// Mitsubishi GX Works2 project: GOL-923VNW-21110019(220112)   PLC: Q02U

PROGRAM OVEN
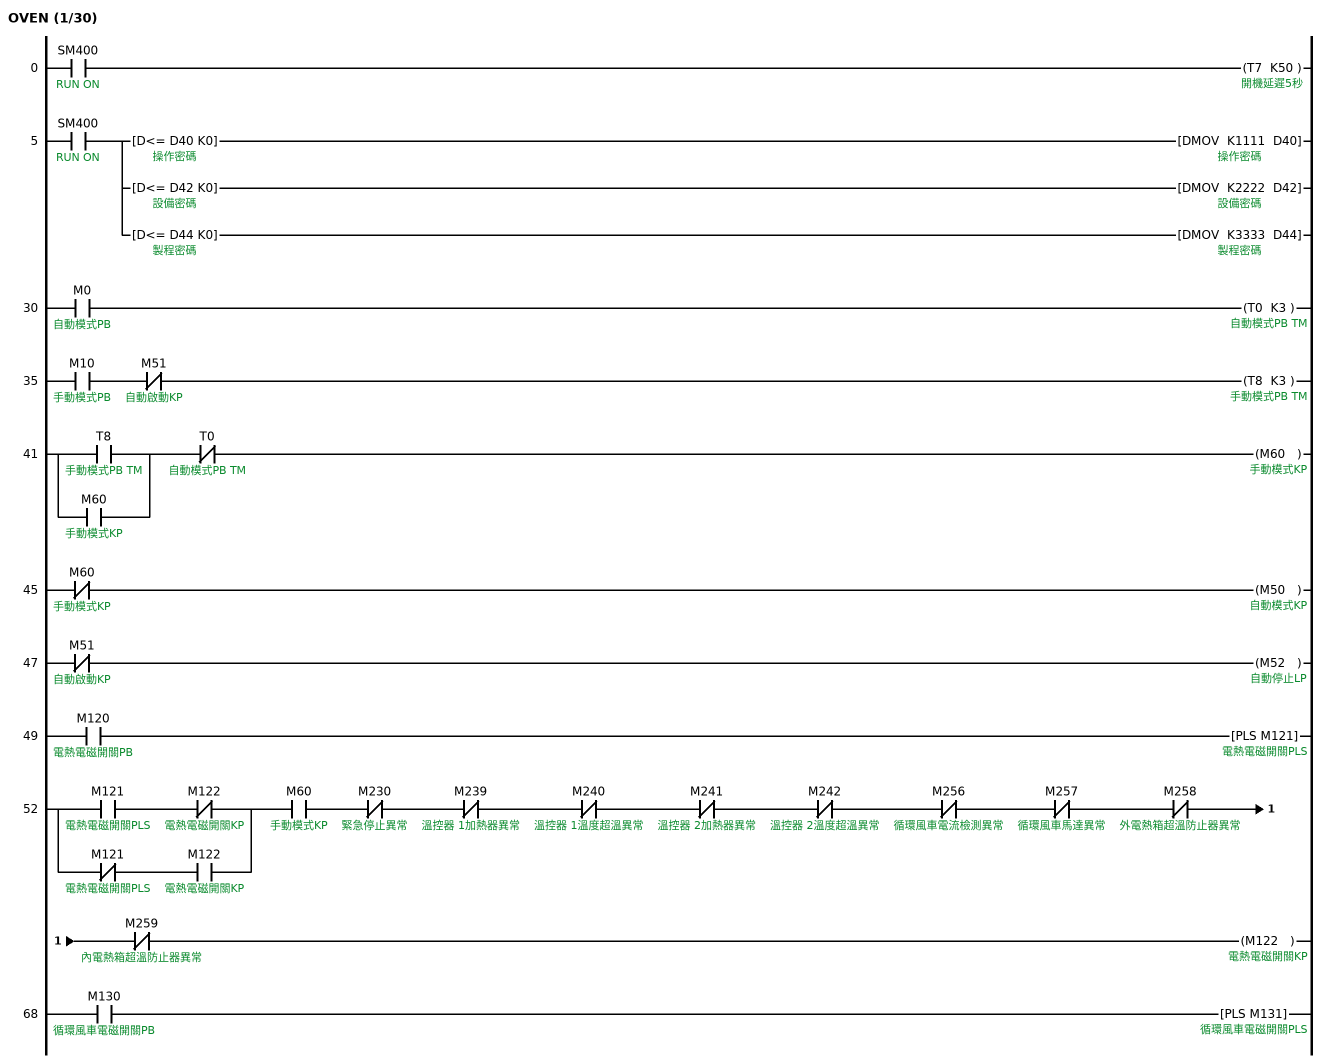
0     LD      SM400  ; RUN ON
      OUT     T7 K50  ; 開機延遲5秒
5     LD      SM400  ; RUN ON
      MPS
      ANDD<=  D40 K0  ; 操作密碼
      DMOV    K1111 D40
      MRD
      ANDD<=  D42 K0  ; 設備密碼
      DMOV    K2222 D42
      MPP
      ANDD<=  D44 K0  ; 製程密碼
      DMOV    K3333 D44
30    LD      M0  ; 自動模式PB
      OUT     T0 K3  ; 自動模式PB TM
35    LD      M10  ; 手動模式PB
      ANI     M51  ; 自動啟動KP
      OUT     T8 K3  ; 手動模式PB TM
41    LD      T8  ; 手動模式PB TM
      OR      M60  ; 手動模式KP
      ANI     T0  ; 自動模式PB TM
      OUT     M60  ; 手動模式KP
45    LDI     M60  ; 手動模式KP
      OUT     M50  ; 自動模式KP
47    LDI     M51  ; 自動啟動KP
      OUT     M52  ; 自動停止LP
49    LD      M120  ; 電熱電磁開關PB
      PLS     M121  ; 電熱電磁開關PLS
52    LD      M121  ; 電熱電磁開關PLS
      ANI     M122  ; 電熱電磁開關KP
      LDI     M121  ; 電熱電磁開關PLS
      AND     M122  ; 電熱電磁開關KP
      ORB
      AND     M60  ; 手動模式KP
      ANI     M230  ; 緊急停止異常
      ANI     M239  ; 溫控器 1加熱器異常
      ANI     M240  ; 溫控器 1溫度超溫異常
      ANI     M241  ; 溫控器 2加熱器異常
      ANI     M242  ; 溫控器 2溫度超溫異常
      ANI     M256  ; 循環風車電流檢測異常
      ANI     M257  ; 循環風車馬達異常
      ANI     M258  ; 外電熱箱超溫防止器異常
      ANI     M259  ; 內電熱箱超溫防止器異常
      OUT     M122  ; 電熱電磁開關KP
68    LD      M130  ; 循環風車電磁開關PB
      PLS     M131  ; 循環風車電磁開關PLS
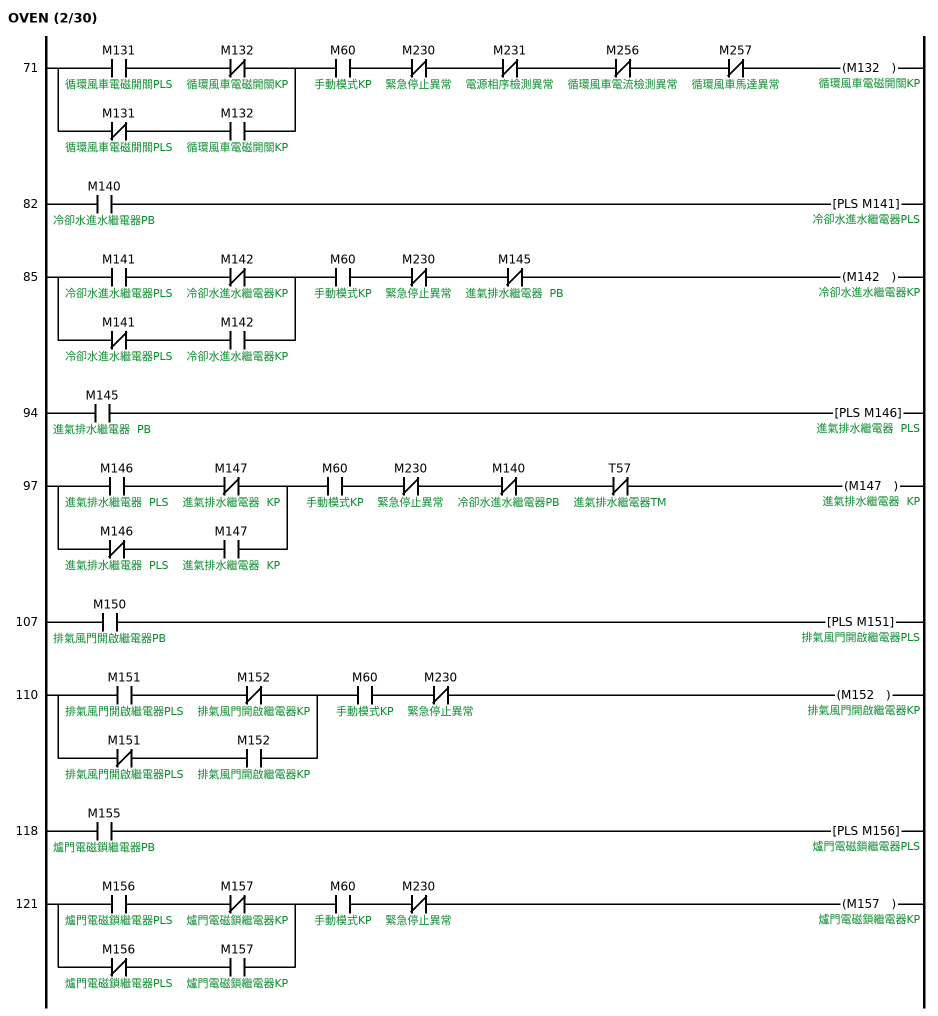
71    LD      M131  ; 循環風車電磁開關PLS
      ANI     M132  ; 循環風車電磁開關KP
      LDI     M131  ; 循環風車電磁開關PLS
      AND     M132  ; 循環風車電磁開關KP
      ORB
      AND     M60  ; 手動模式KP
      ANI     M230  ; 緊急停止異常
      ANI     M231  ; 電源相序檢測異常
      ANI     M256  ; 循環風車電流檢測異常
      ANI     M257  ; 循環風車馬達異常
      OUT     M132  ; 循環風車電磁開關KP
82    LD      M140  ; 冷卻水進水繼電器PB
      PLS     M141  ; 冷卻水進水繼電器PLS
85    LD      M141  ; 冷卻水進水繼電器PLS
      ANI     M142  ; 冷卻水進水繼電器KP
      LDI     M141  ; 冷卻水進水繼電器PLS
      AND     M142  ; 冷卻水進水繼電器KP
      ORB
      AND     M60  ; 手動模式KP
      ANI     M230  ; 緊急停止異常
      ANI     M145  ; 進氣排水繼電器  PB
      OUT     M142  ; 冷卻水進水繼電器KP
94    LD      M145  ; 進氣排水繼電器  PB
      PLS     M146  ; 進氣排水繼電器  PLS
97    LD      M146  ; 進氣排水繼電器  PLS
      ANI     M147  ; 進氣排水繼電器  KP
      LDI     M146  ; 進氣排水繼電器  PLS
      AND     M147  ; 進氣排水繼電器  KP
      ORB
      AND     M60  ; 手動模式KP
      ANI     M230  ; 緊急停止異常
      ANI     M140  ; 冷卻水進水繼電器PB
      ANI     T57  ; 進氣排水繼電器TM
      OUT     M147  ; 進氣排水繼電器  KP
107   LD      M150  ; 排氣風門開啟繼電器PB
      PLS     M151  ; 排氣風門開啟繼電器PLS
110   LD      M151  ; 排氣風門開啟繼電器PLS
      ANI     M152  ; 排氣風門開啟繼電器KP
      LDI     M151  ; 排氣風門開啟繼電器PLS
      AND     M152  ; 排氣風門開啟繼電器KP
      ORB
      AND     M60  ; 手動模式KP
      ANI     M230  ; 緊急停止異常
      OUT     M152  ; 排氣風門開啟繼電器KP
118   LD      M155  ; 爐門電磁鎖繼電器PB
      PLS     M156  ; 爐門電磁鎖繼電器PLS
121   LD      M156  ; 爐門電磁鎖繼電器PLS
      ANI     M157  ; 爐門電磁鎖繼電器KP
      LDI     M156  ; 爐門電磁鎖繼電器PLS
      AND     M157  ; 爐門電磁鎖繼電器KP
      ORB
      AND     M60  ; 手動模式KP
      ANI     M230  ; 緊急停止異常
      OUT     M157  ; 爐門電磁鎖繼電器KP
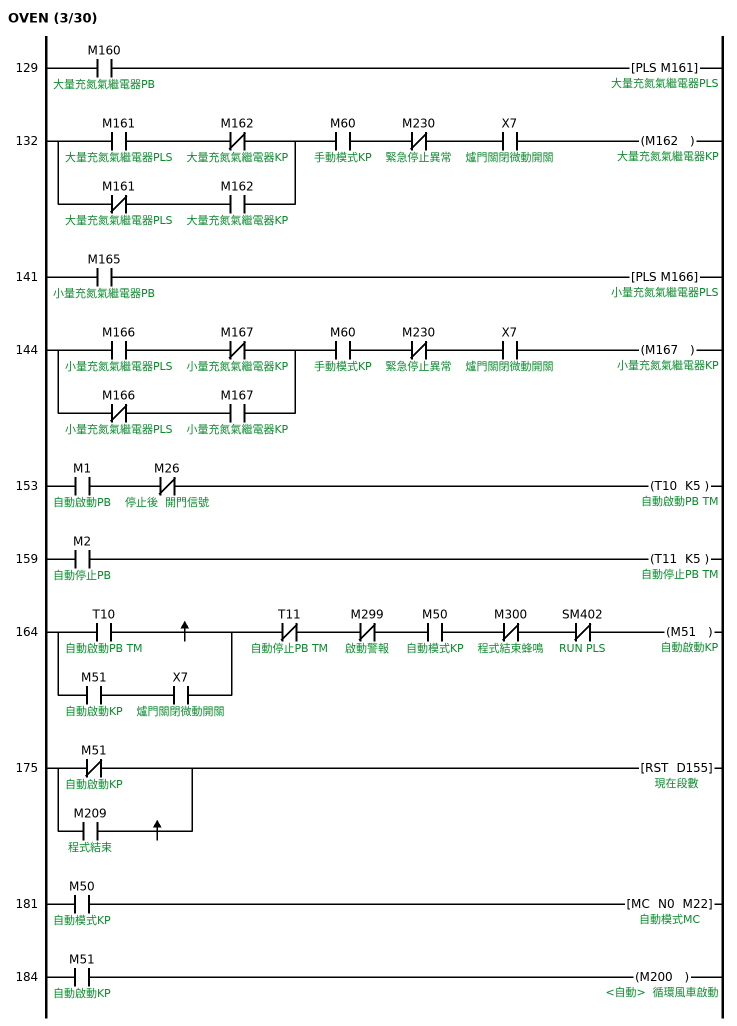
129   LD      M160  ; 大量充氮氣繼電器PB
      PLS     M161  ; 大量充氮氣繼電器PLS
132   LD      M161  ; 大量充氮氣繼電器PLS
      ANI     M162  ; 大量充氮氣繼電器KP
      LDI     M161  ; 大量充氮氣繼電器PLS
      AND     M162  ; 大量充氮氣繼電器KP
      ORB
      AND     M60  ; 手動模式KP
      ANI     M230  ; 緊急停止異常
      AND     X7  ; 爐門關閉微動開關
      OUT     M162  ; 大量充氮氣繼電器KP
141   LD      M165  ; 小量充氮氣繼電器PB
      PLS     M166  ; 小量充氮氣繼電器PLS
144   LD      M166  ; 小量充氮氣繼電器PLS
      ANI     M167  ; 小量充氮氣繼電器KP
      LDI     M166  ; 小量充氮氣繼電器PLS
      AND     M167  ; 小量充氮氣繼電器KP
      ORB
      AND     M60  ; 手動模式KP
      ANI     M230  ; 緊急停止異常
      AND     X7  ; 爐門關閉微動開關
      OUT     M167  ; 小量充氮氣繼電器KP
153   LD      M1  ; 自動啟動PB
      ANI     M26  ; 停止後  開門信號
      OUT     T10 K5  ; 自動啟動PB TM
159   LD      M2  ; 自動停止PB
      OUT     T11 K5  ; 自動停止PB TM
164   LD      T10  ; 自動啟動PB TM
      MEP
      LD      M51  ; 自動啟動KP
      AND     X7  ; 爐門關閉微動開關
      ORB
      ANI     T11  ; 自動停止PB TM
      ANI     M299  ; 啟動警報
      AND     M50  ; 自動模式KP
      ANI     M300  ; 程式結束蜂鳴
      ANI     SM402  ; RUN PLS
      OUT     M51  ; 自動啟動KP
175   LDI     M51  ; 自動啟動KP
      LD      M209  ; 程式結束
      MEP
      ORB
      RST     D155  ; 現在段數
181   LD      M50  ; 自動模式KP
      MC      N0 M22  ; 自動模式MC
184   LD      M51  ; 自動啟動KP
      OUT     M200  ; <自動>  循環風車啟動
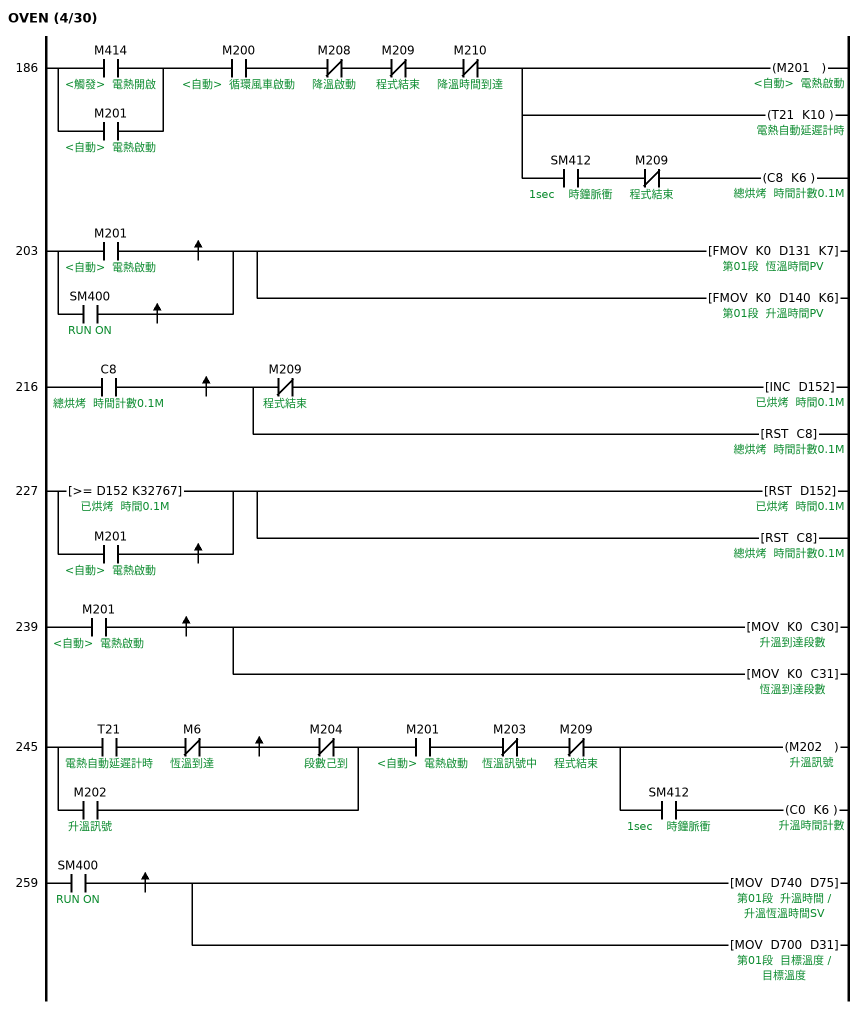
186   LD      M414  ; <觸發>  電熱開啟
      OR      M201  ; <自動>  電熱啟動
      AND     M200  ; <自動>  循環風車啟動
      ANI     M208  ; 降溫啟動
      ANI     M209  ; 程式結束
      ANI     M210  ; 降溫時間到達
      OUT     M201  ; <自動>  電熱啟動
      OUT     T21 K10  ; 電熱自動延遲計時
      AND     SM412  ; 1sec    時鐘脈衝
      ANI     M209  ; 程式結束
      OUT     C8 K6  ; 總烘烤  時間計數0.1M
203   LD      M201  ; <自動>  電熱啟動
      MEP
      LD      SM400  ; RUN ON
      MEP
      ORB
      FMOV    K0 D131 K7  ; 第01段  恆溫時間PV
      FMOV    K0 D140 K6  ; 第01段  升溫時間PV
216   LD      C8  ; 總烘烤  時間計數0.1M
      MEP
      MPS
      ANI     M209  ; 程式結束
      INC     D152  ; 已烘烤  時間0.1M
      MPP
      RST     C8  ; 總烘烤  時間計數0.1M
227   LD>=    D152 K32767  ; 已烘烤  時間0.1M
      LD      M201  ; <自動>  電熱啟動
      MEP
      ORB
      RST     D152  ; 已烘烤  時間0.1M
      RST     C8  ; 總烘烤  時間計數0.1M
239   LD      M201  ; <自動>  電熱啟動
      MEP
      MOV     K0 C30  ; 升溫到達段數
      MOV     K0 C31  ; 恆溫到達段數
245   LD      T21  ; 電熱自動延遲計時
      ANI     M6  ; 恆溫到達
      MEP
      ANI     M204  ; 段數己到
      OR      M202  ; 升溫訊號
      AND     M201  ; <自動>  電熱啟動
      ANI     M203  ; 恆溫訊號中
      ANI     M209  ; 程式結束
      OUT     M202  ; 升溫訊號
      AND     SM412  ; 1sec    時鐘脈衝
      OUT     C0 K6  ; 升溫時間計數
259   LD      SM400  ; RUN ON
      MEP
      MOV     D740 D75  ; 第01段  升溫時間 / 升溫恆溫時間SV
      MOV     D700 D31  ; 第01段  目標溫度 / 目標溫度
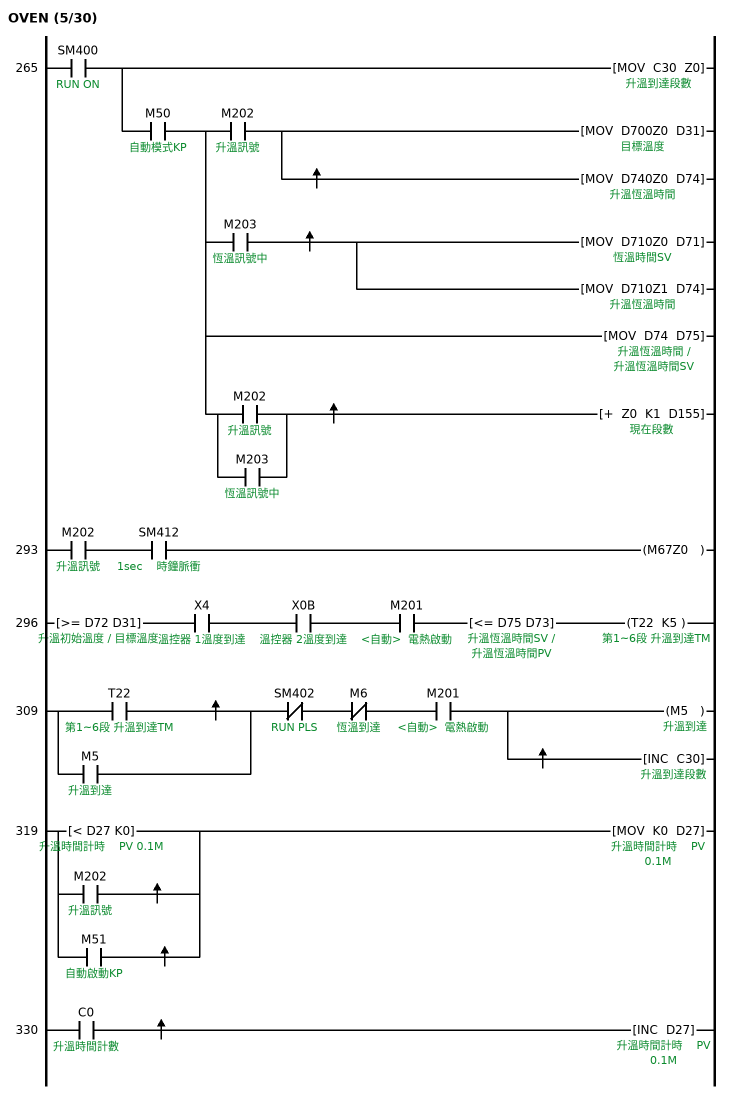
265   LD      SM400  ; RUN ON
      MOV     C30 Z0
      AND     M50  ; 自動模式KP
      MPS
      AND     M202  ; 升溫訊號
      MOV     D700Z0 D31
      MEP
      MOV     D740Z0 D74  ; 升溫恆溫時間
      MRD
      AND     M203  ; 恆溫訊號中
      MEP
      MOV     D710Z0 D71  ; 恆溫時間SV
      MOV     D710Z1 D74
      MPP
      MOV     D74 D75
      LD      M202  ; 升溫訊號
      OR      M203  ; 恆溫訊號中
      ANB
      MEP
      +       Z0 K1 D155
293   LD      M202  ; 升溫訊號
      AND     SM412  ; 1sec    時鐘脈衝
      OUT     M67Z0
296   LD>=    D72 D31  ; 升溫初始溫度 / 目標溫度
      AND     X4  ; 溫控器 1溫度到達
      AND     X0B  ; 溫控器 2溫度到達
      AND     M201  ; <自動>  電熱啟動
      AND<=   D75 D73  ; 升溫恆溫時間SV / 升溫恆溫時間PV
      OUT     T22 K5  ; 第1~6段 升溫到達TM
309   LD      T22  ; 第1~6段 升溫到達TM
      MEP
      OR      M5  ; 升溫到達
      ANI     SM402  ; RUN PLS
      ANI     M6  ; 恆溫到達
      AND     M201  ; <自動>  電熱啟動
      OUT     M5  ; 升溫到達
      MEP
      INC     C30
319   LD<     D27 K0  ; 升溫時間計時    PV 0.1M
      LD      M202  ; 升溫訊號
      MEP
      ORB
      LD      M51  ; 自動啟動KP
      MEP
      ORB
      MOV     K0 D27
330   LD      C0  ; 升溫時間計數
      MEP
      INC     D27
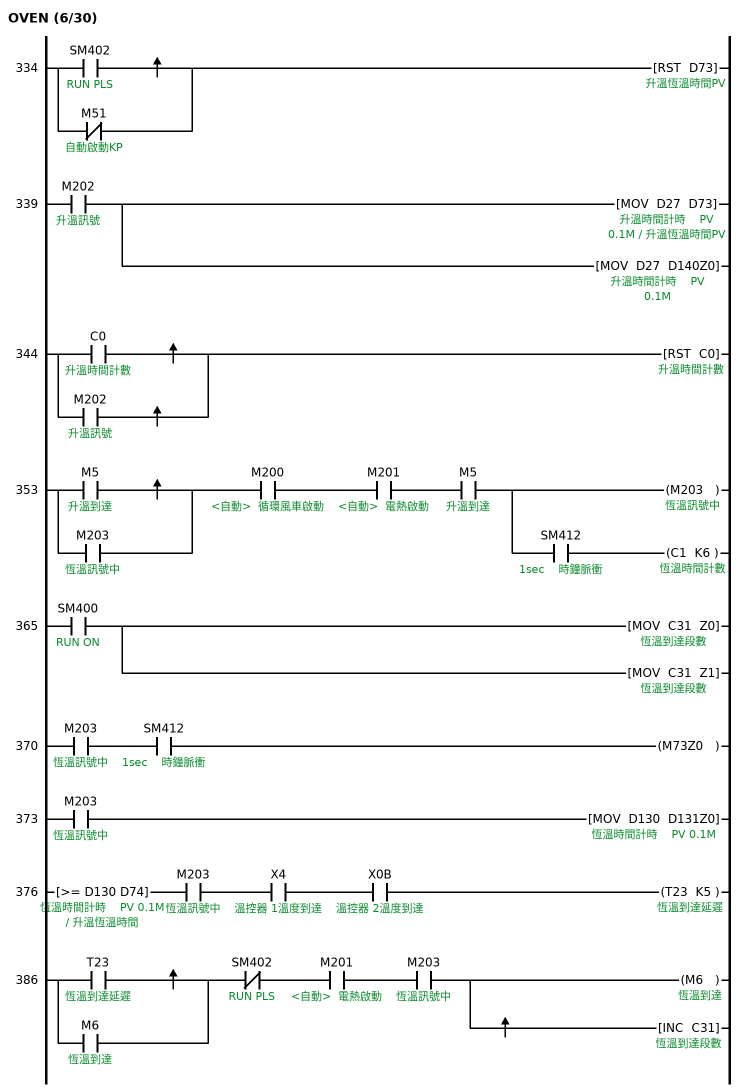
334   LD      SM402  ; RUN PLS
      MEP
      ORI     M51  ; 自動啟動KP
      RST     D73  ; 升溫恆溫時間PV
339   LD      M202  ; 升溫訊號
      MOV     D27 D73
      MOV     D27 D140Z0
344   LD      C0  ; 升溫時間計數
      MEP
      LD      M202  ; 升溫訊號
      MEP
      ORB
      RST     C0  ; 升溫時間計數
353   LD      M5  ; 升溫到達
      MEP
      OR      M203  ; 恆溫訊號中
      AND     M200  ; <自動>  循環風車啟動
      AND     M201  ; <自動>  電熱啟動
      AND     M5  ; 升溫到達
      OUT     M203  ; 恆溫訊號中
      AND     SM412  ; 1sec    時鐘脈衝
      OUT     C1 K6  ; 恆溫時間計數
365   LD      SM400  ; RUN ON
      MOV     C31 Z0
      MOV     C31 Z1
370   LD      M203  ; 恆溫訊號中
      AND     SM412  ; 1sec    時鐘脈衝
      OUT     M73Z0
373   LD      M203  ; 恆溫訊號中
      MOV     D130 D131Z0  ; 恆溫時間計時    PV 0.1M
376   LD>=    D130 D74  ; 恆溫時間計時    PV 0.1M / 升溫恆溫時間
      AND     M203  ; 恆溫訊號中
      AND     X4  ; 溫控器 1溫度到達
      AND     X0B  ; 溫控器 2溫度到達
      OUT     T23 K5  ; 恆溫到達延遲
386   LD      T23  ; 恆溫到達延遲
      MEP
      OR      M6  ; 恆溫到達
      ANI     SM402  ; RUN PLS
      AND     M201  ; <自動>  電熱啟動
      AND     M203  ; 恆溫訊號中
      OUT     M6  ; 恆溫到達
      MEP
      INC     C31
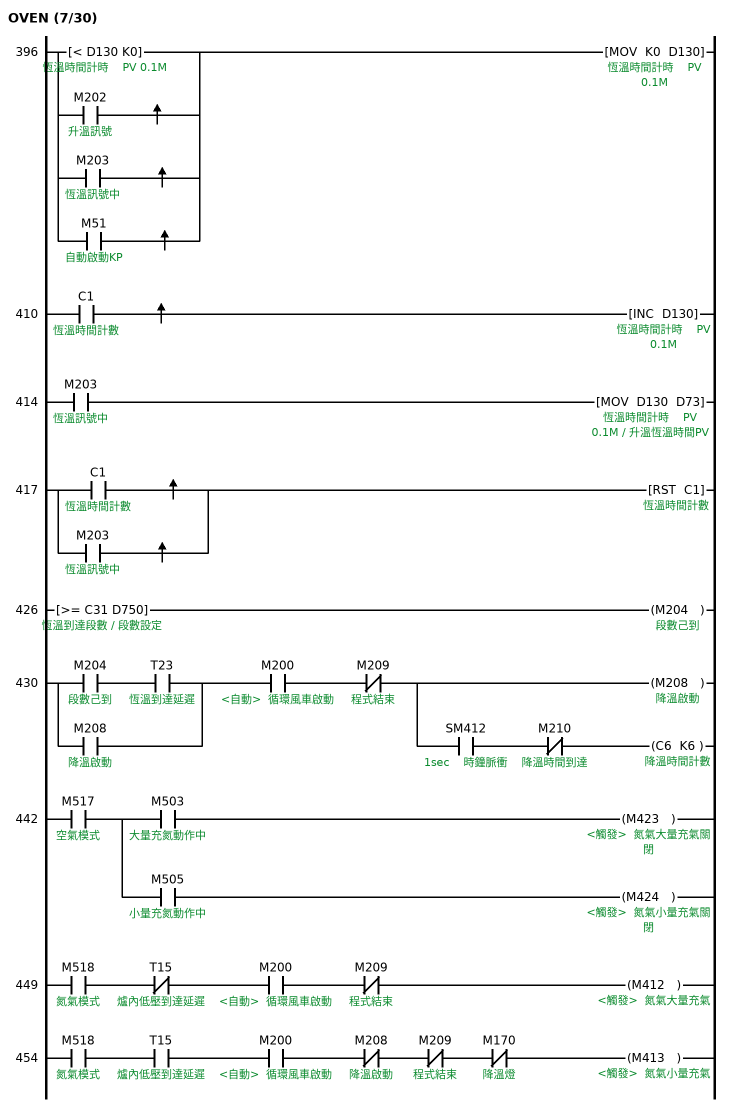
396   LD<     D130 K0  ; 恆溫時間計時    PV 0.1M
      LD      M202  ; 升溫訊號
      MEP
      ORB
      LD      M203  ; 恆溫訊號中
      MEP
      ORB
      LD      M51  ; 自動啟動KP
      MEP
      ORB
      MOV     K0 D130
410   LD      C1  ; 恆溫時間計數
      MEP
      INC     D130
414   LD      M203  ; 恆溫訊號中
      MOV     D130 D73
417   LD      C1  ; 恆溫時間計數
      MEP
      LD      M203  ; 恆溫訊號中
      MEP
      ORB
      RST     C1  ; 恆溫時間計數
426   LD>=    C31 D750  ; 恆溫到達段數 / 段數設定
      OUT     M204  ; 段數己到
430   LD      M204  ; 段數己到
      AND     T23  ; 恆溫到達延遲
      OR      M208  ; 降溫啟動
      AND     M200  ; <自動>  循環風車啟動
      ANI     M209  ; 程式結束
      OUT     M208  ; 降溫啟動
      AND     SM412  ; 1sec    時鐘脈衝
      ANI     M210  ; 降溫時間到達
      OUT     C6 K6  ; 降溫時間計數
442   LD      M517  ; 空氣模式
      MPS
      AND     M503  ; 大量充氮動作中
      OUT     M423  ; <觸發>  氮氣大量充氣關閉
      MPP
      AND     M505  ; 小量充氮動作中
      OUT     M424  ; <觸發>  氮氣小量充氣關閉
449   LD      M518  ; 氮氣模式
      ANI     T15  ; 爐內低壓到達延遲
      AND     M200  ; <自動>  循環風車啟動
      ANI     M209  ; 程式結束
      OUT     M412  ; <觸發>  氮氣大量充氣
454   LD      M518  ; 氮氣模式
      AND     T15  ; 爐內低壓到達延遲
      AND     M200  ; <自動>  循環風車啟動
      ANI     M208  ; 降溫啟動
      ANI     M209  ; 程式結束
      ANI     M170  ; 降溫燈
      OUT     M413  ; <觸發>  氮氣小量充氣
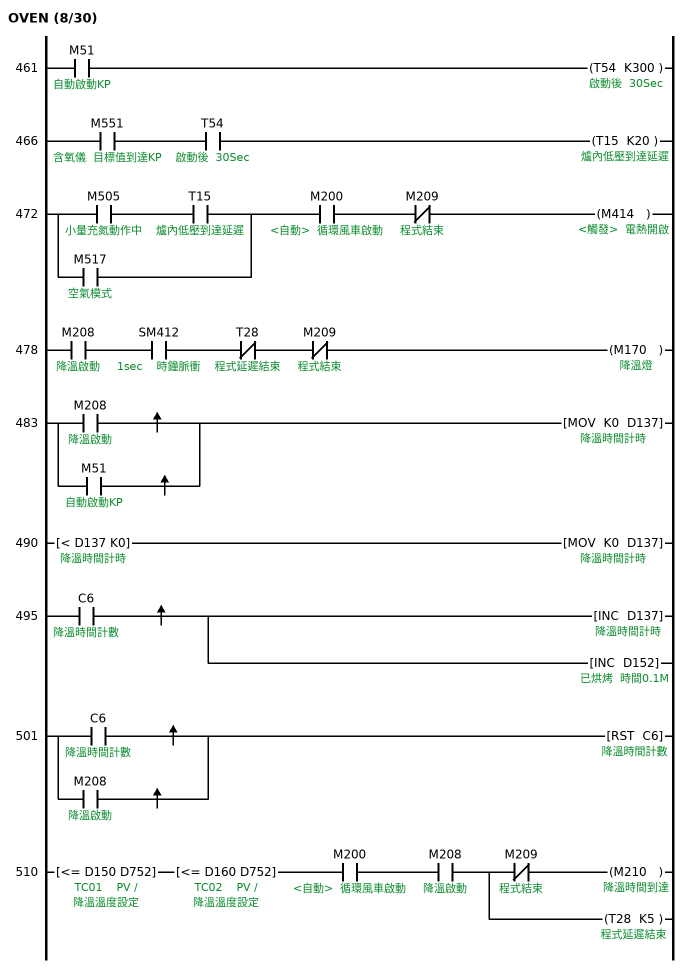
461   LD      M51  ; 自動啟動KP
      OUT     T54 K300  ; 啟動後  30Sec
466   LD      M551  ; 含氧儀  目標值到達KP
      AND     T54  ; 啟動後  30Sec
      OUT     T15 K20  ; 爐內低壓到達延遲
472   LD      M505  ; 小量充氮動作中
      AND     T15  ; 爐內低壓到達延遲
      OR      M517  ; 空氣模式
      AND     M200  ; <自動>  循環風車啟動
      ANI     M209  ; 程式結束
      OUT     M414  ; <觸發>  電熱開啟
478   LD      M208  ; 降溫啟動
      AND     SM412  ; 1sec    時鐘脈衝
      ANI     T28  ; 程式延遲結束
      ANI     M209  ; 程式結束
      OUT     M170  ; 降溫燈
483   LD      M208  ; 降溫啟動
      MEP
      LD      M51  ; 自動啟動KP
      MEP
      ORB
      MOV     K0 D137  ; 降溫時間計時
490   LD<     D137 K0  ; 降溫時間計時
      MOV     K0 D137
495   LD      C6  ; 降溫時間計數
      MEP
      INC     D137
      INC     D152
501   LD      C6  ; 降溫時間計數
      MEP
      LD      M208  ; 降溫啟動
      MEP
      ORB
      RST     C6  ; 降溫時間計數
510   LD<=    D150 D752  ; TC01    PV / 降溫溫度設定
      AND<=   D160 D752  ; TC02    PV / 降溫溫度設定
      AND     M200  ; <自動>  循環風車啟動
      AND     M208  ; 降溫啟動
      MPS
      ANI     M209  ; 程式結束
      OUT     M210  ; 降溫時間到達
      MPP
      OUT     T28 K5  ; 程式延遲結束
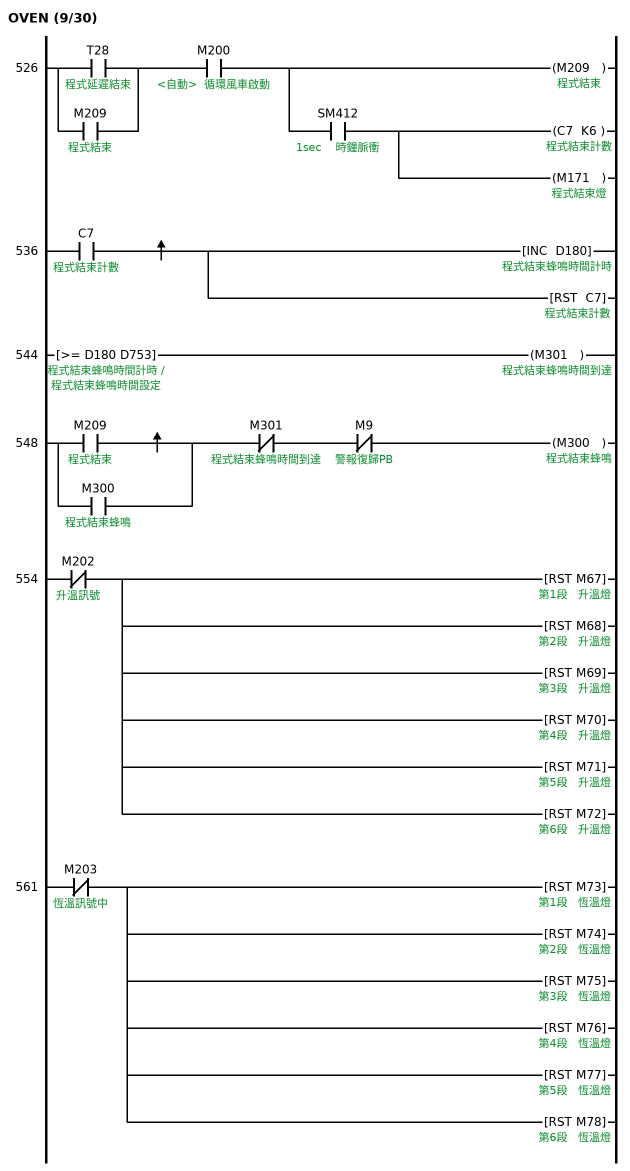
526   LD      T28  ; 程式延遲結束
      OR      M209  ; 程式結束
      AND     M200  ; <自動>  循環風車啟動
      OUT     M209  ; 程式結束
      AND     SM412  ; 1sec    時鐘脈衝
      OUT     C7 K6  ; 程式結束計數
      OUT     M171  ; 程式結束燈
536   LD      C7  ; 程式結束計數
      MEP
      INC     D180  ; 程式結束蜂鳴時間計時
      RST     C7  ; 程式結束計數
544   LD>=    D180 D753  ; 程式結束蜂鳴時間計時 / 程式結束蜂鳴時間設定
      OUT     M301  ; 程式結束蜂鳴時間到達
548   LD      M209  ; 程式結束
      MEP
      OR      M300  ; 程式結束蜂鳴
      ANI     M301  ; 程式結束蜂鳴時間到達
      ANI     M9  ; 警報復歸PB
      OUT     M300  ; 程式結束蜂鳴
554   LDI     M202  ; 升溫訊號
      RST     M67  ; 第1段   升溫燈
      RST     M68  ; 第2段   升溫燈
      RST     M69  ; 第3段   升溫燈
      RST     M70  ; 第4段   升溫燈
      RST     M71  ; 第5段   升溫燈
      RST     M72  ; 第6段   升溫燈
561   LDI     M203  ; 恆溫訊號中
      RST     M73  ; 第1段   恆溫燈
      RST     M74  ; 第2段   恆溫燈
      RST     M75  ; 第3段   恆溫燈
      RST     M76  ; 第4段   恆溫燈
      RST     M77  ; 第5段   恆溫燈
      RST     M78  ; 第6段   恆溫燈
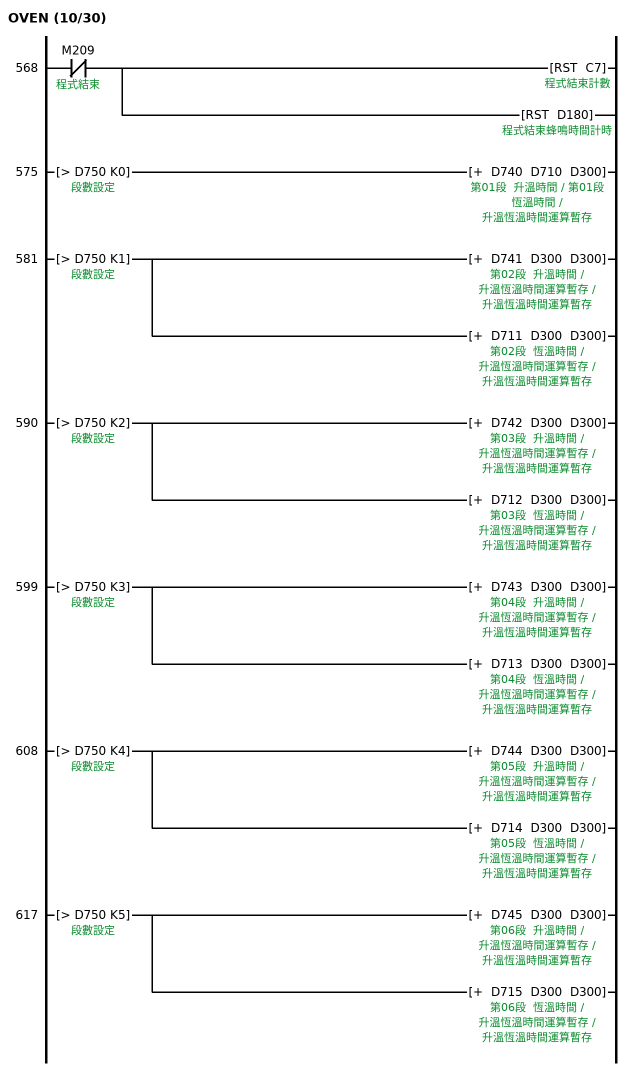
568   LDI     M209  ; 程式結束
      RST     C7  ; 程式結束計數
      RST     D180  ; 程式結束蜂鳴時間計時
575   LD>     D750 K0  ; 段數設定
      +       D740 D710 D300  ; 第01段  恆溫時間 / 升溫恆溫時間運算暫存
581   LD>     D750 K1  ; 段數設定
      +       D741 D300 D300  ; 第02段  升溫時間
      +       D711 D300 D300  ; 第02段  恆溫時間
590   LD>     D750 K2  ; 段數設定
      +       D742 D300 D300  ; 第03段  升溫時間
      +       D712 D300 D300  ; 第03段  恆溫時間
599   LD>     D750 K3  ; 段數設定
      +       D743 D300 D300  ; 第04段  升溫時間
      +       D713 D300 D300  ; 第04段  恆溫時間
608   LD>     D750 K4  ; 段數設定
      +       D744 D300 D300  ; 第05段  升溫時間
      +       D714 D300 D300  ; 第05段  恆溫時間
617   LD>     D750 K5  ; 段數設定
      +       D745 D300 D300  ; 第06段  升溫時間
      +       D715 D300 D300  ; 第06段  恆溫時間
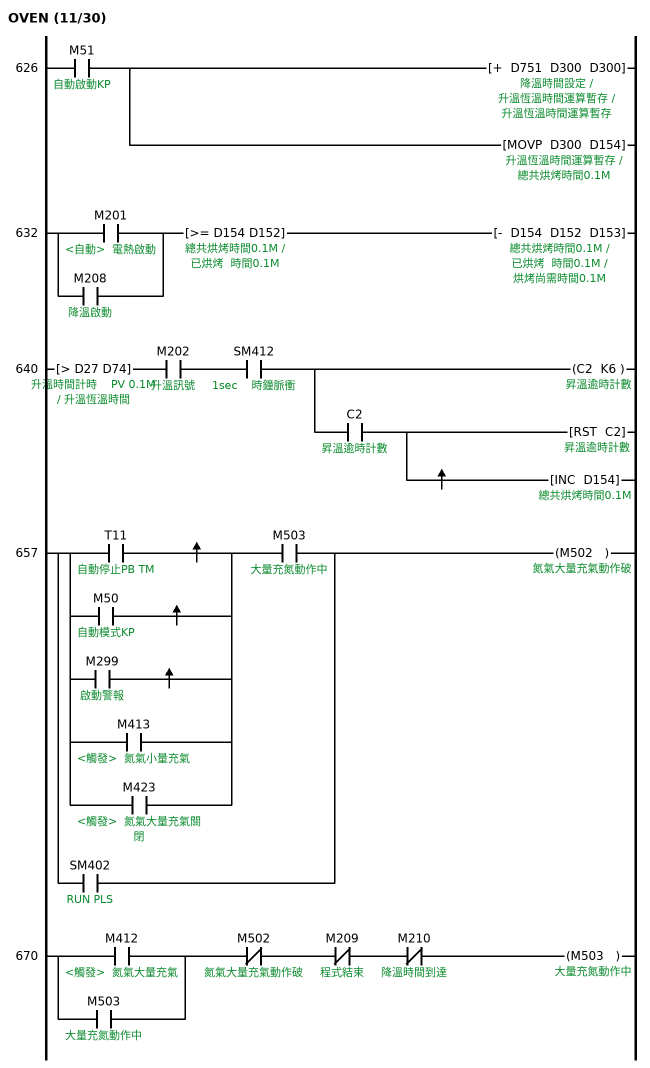
626   LD      M51  ; 自動啟動KP
      +       D751 D300 D300  ; 降溫時間設定
      MOVP    D300 D154  ; 總共烘烤時間0.1M
632   LD      M201  ; <自動>  電熱啟動
      OR      M208  ; 降溫啟動
      AND>=   D154 D152  ; 總共烘烤時間0.1M / 已烘烤  時間0.1M
      -       D154 D152 D153  ; 烘烤尚需時間0.1M
640   LD>     D27 D74  ; 升溫時間計時    PV 0.1M / 升溫恆溫時間
      AND     M202  ; 升溫訊號
      AND     SM412  ; 1sec    時鐘脈衝
      OUT     C2 K6  ; 昇溫逾時計數
      AND     C2  ; 昇溫逾時計數
      RST     C2  ; 昇溫逾時計數
      MEP
      INC     D154
657   LD      T11  ; 自動停止PB TM
      MEP
      LD      M50  ; 自動模式KP
      MEP
      ORB
      LD      M299  ; 啟動警報
      MEP
      ORB
      OR      M413  ; <觸發>  氮氣小量充氣
      OR      M423  ; <觸發>  氮氣大量充氣關閉
      AND     M503  ; 大量充氮動作中
      OR      SM402  ; RUN PLS
      OUT     M502  ; 氮氣大量充氣動作破
670   LD      M412  ; <觸發>  氮氣大量充氣
      OR      M503  ; 大量充氮動作中
      ANI     M502  ; 氮氣大量充氣動作破
      ANI     M209  ; 程式結束
      ANI     M210  ; 降溫時間到達
      OUT     M503  ; 大量充氮動作中
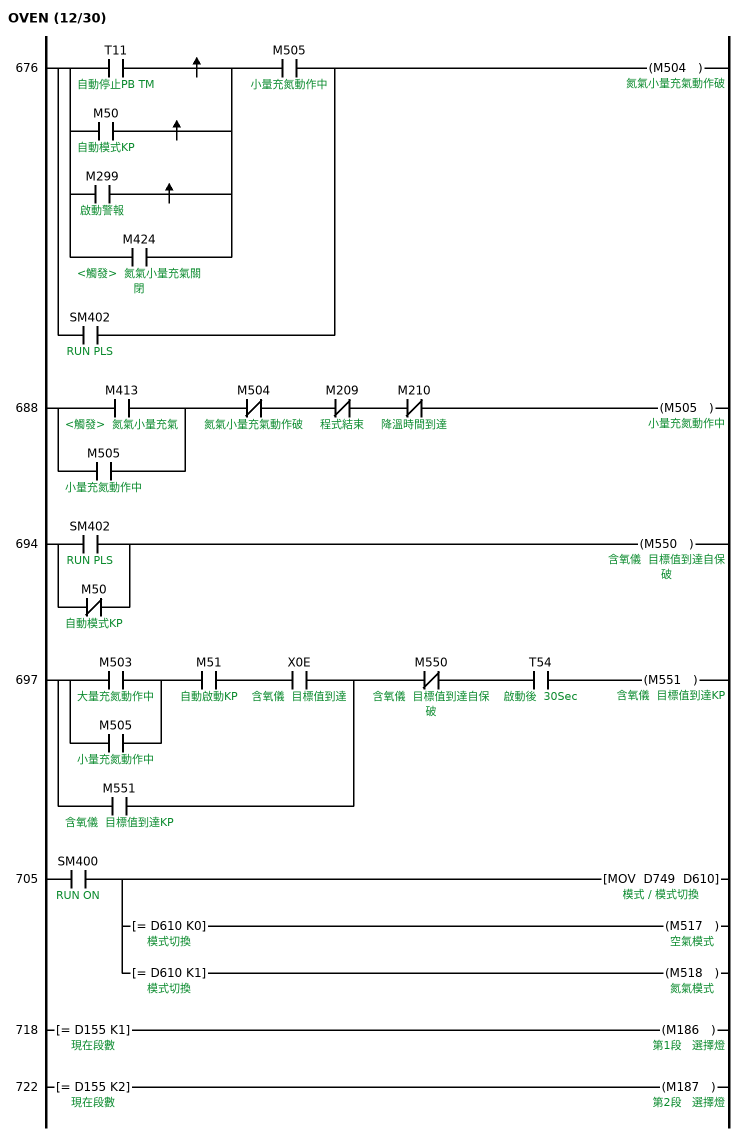
676   LD      T11  ; 自動停止PB TM
      MEP
      LD      M50  ; 自動模式KP
      MEP
      ORB
      LD      M299  ; 啟動警報
      MEP
      ORB
      OR      M424  ; <觸發>  氮氣小量充氣關閉
      AND     M505  ; 小量充氮動作中
      OR      SM402  ; RUN PLS
      OUT     M504  ; 氮氣小量充氣動作破
688   LD      M413  ; <觸發>  氮氣小量充氣
      OR      M505  ; 小量充氮動作中
      ANI     M504  ; 氮氣小量充氣動作破
      ANI     M209  ; 程式結束
      ANI     M210  ; 降溫時間到達
      OUT     M505  ; 小量充氮動作中
694   LD      SM402  ; RUN PLS
      ORI     M50  ; 自動模式KP
      OUT     M550  ; 含氧儀  目標值到達自保破
697   LD      M503  ; 大量充氮動作中
      OR      M505  ; 小量充氮動作中
      AND     M51  ; 自動啟動KP
      AND     X0E  ; 含氧儀  目標值到達
      OR      M551  ; 含氧儀  目標值到達KP
      ANI     M550  ; 含氧儀  目標值到達自保破
      AND     T54  ; 啟動後  30Sec
      OUT     M551  ; 含氧儀  目標值到達KP
705   LD      SM400  ; RUN ON
      MOV     D749 D610  ; 模式 / 模式切換
      MPS
      AND=    D610 K0  ; 模式切換
      OUT     M517  ; 空氣模式
      MPP
      AND=    D610 K1  ; 模式切換
      OUT     M518  ; 氮氣模式
718   LD=     D155 K1  ; 現在段數
      OUT     M186  ; 第1段   選擇燈
722   LD=     D155 K2  ; 現在段數
      OUT     M187  ; 第2段   選擇燈
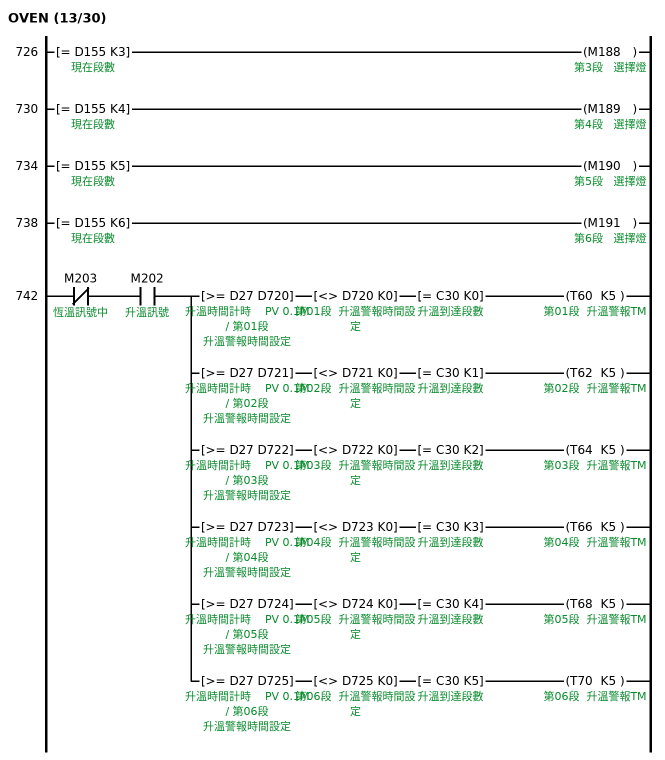
726   LD=     D155 K3  ; 現在段數
      OUT     M188  ; 第3段   選擇燈
730   LD=     D155 K4  ; 現在段數
      OUT     M189  ; 第4段   選擇燈
734   LD=     D155 K5  ; 現在段數
      OUT     M190  ; 第5段   選擇燈
738   LD=     D155 K6  ; 現在段數
      OUT     M191  ; 第6段   選擇燈
742   LDI     M203  ; 恆溫訊號中
      AND     M202  ; 升溫訊號
      MPS
      AND>=   D27 D720  ; 升溫時間計時    PV 0.1M / 第01段  升溫警報時間設定
      AND<>   D720 K0  ; 第01段  升溫警報時間設定
      AND=    C30 K0  ; 升溫到達段數
      OUT     T60 K5  ; 第01段  升溫警報TM
      MRD
      AND>=   D27 D721  ; 升溫時間計時    PV 0.1M / 第02段  升溫警報時間設定
      AND<>   D721 K0  ; 第02段  升溫警報時間設定
      AND=    C30 K1  ; 升溫到達段數
      OUT     T62 K5  ; 第02段  升溫警報TM
      MRD
      AND>=   D27 D722  ; 升溫時間計時    PV 0.1M / 第03段  升溫警報時間設定
      AND<>   D722 K0  ; 第03段  升溫警報時間設定
      AND=    C30 K2  ; 升溫到達段數
      OUT     T64 K5  ; 第03段  升溫警報TM
      MRD
      AND>=   D27 D723  ; 升溫時間計時    PV 0.1M / 第04段  升溫警報時間設定
      AND<>   D723 K0  ; 第04段  升溫警報時間設定
      AND=    C30 K3  ; 升溫到達段數
      OUT     T66 K5  ; 第04段  升溫警報TM
      MRD
      AND>=   D27 D724  ; 升溫時間計時    PV 0.1M / 第05段  升溫警報時間設定
      AND<>   D724 K0  ; 第05段  升溫警報時間設定
      AND=    C30 K4  ; 升溫到達段數
      OUT     T68 K5  ; 第05段  升溫警報TM
      MPP
      AND>=   D27 D725  ; 升溫時間計時    PV 0.1M / 第06段  升溫警報時間設定
      AND<>   D725 K0  ; 第06段  升溫警報時間設定
      AND=    C30 K5  ; 升溫到達段數
      OUT     T70 K5  ; 第06段  升溫警報TM
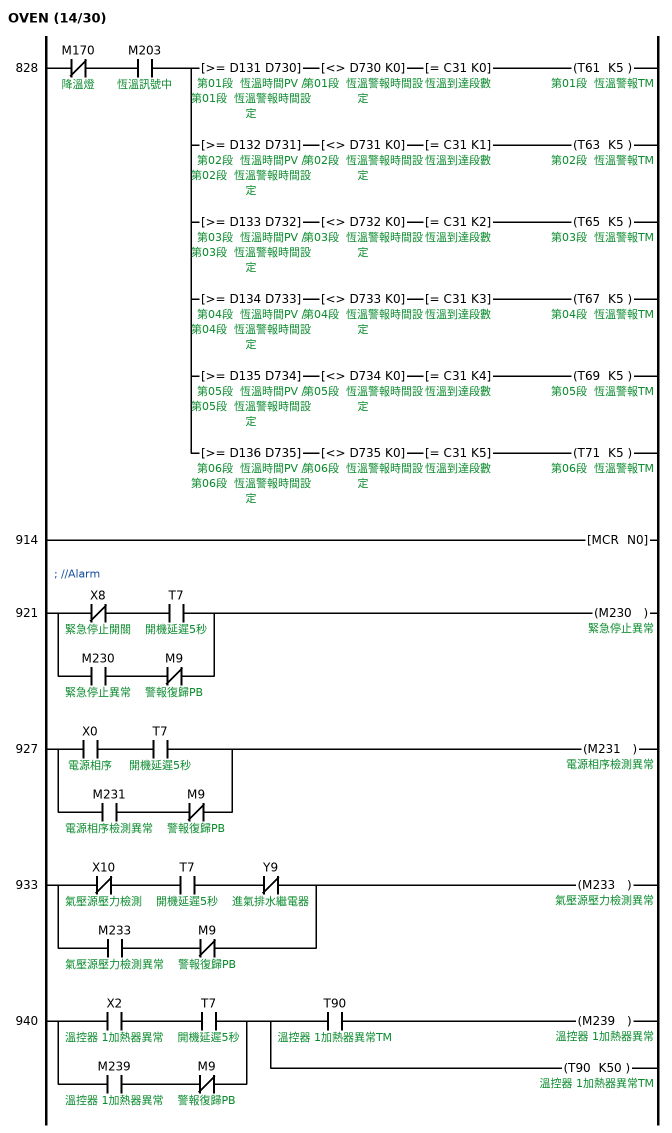
828   LDI     M170  ; 降溫燈
      AND     M203  ; 恆溫訊號中
      MPS
      AND>=   D131 D730  ; 第01段  恆溫時間PV / 第01段  恆溫警報時間設定
      AND<>   D730 K0  ; 第01段  恆溫警報時間設定
      AND=    C31 K0  ; 恆溫到達段數
      OUT     T61 K5  ; 第01段  恆溫警報TM
      MRD
      AND>=   D132 D731  ; 第02段  恆溫時間PV / 第02段  恆溫警報時間設定
      AND<>   D731 K0  ; 第02段  恆溫警報時間設定
      AND=    C31 K1  ; 恆溫到達段數
      OUT     T63 K5  ; 第02段  恆溫警報TM
      MRD
      AND>=   D133 D732  ; 第03段  恆溫時間PV / 第03段  恆溫警報時間設定
      AND<>   D732 K0  ; 第03段  恆溫警報時間設定
      AND=    C31 K2  ; 恆溫到達段數
      OUT     T65 K5  ; 第03段  恆溫警報TM
      MRD
      AND>=   D134 D733  ; 第04段  恆溫時間PV / 第04段  恆溫警報時間設定
      AND<>   D733 K0  ; 第04段  恆溫警報時間設定
      AND=    C31 K3  ; 恆溫到達段數
      OUT     T67 K5  ; 第04段  恆溫警報TM
      MRD
      AND>=   D135 D734  ; 第05段  恆溫時間PV / 第05段  恆溫警報時間設定
      AND<>   D734 K0  ; 第05段  恆溫警報時間設定
      AND=    C31 K4  ; 恆溫到達段數
      OUT     T69 K5  ; 第05段  恆溫警報TM
      MPP
      AND>=   D136 D735  ; 第06段  恆溫時間PV / 第06段  恆溫警報時間設定
      AND<>   D735 K0  ; 第06段  恆溫警報時間設定
      AND=    C31 K5  ; 恆溫到達段數
      OUT     T71 K5  ; 第06段  恆溫警報TM
914   MCR     N0
; //Alarm
921   LDI     X8  ; 緊急停止開關
      AND     T7  ; 開機延遲5秒
      LD      M230  ; 緊急停止異常
      ANI     M9  ; 警報復歸PB
      ORB
      OUT     M230  ; 緊急停止異常
927   LD      X0  ; 電源相序
      AND     T7  ; 開機延遲5秒
      LD      M231  ; 電源相序檢測異常
      ANI     M9  ; 警報復歸PB
      ORB
      OUT     M231  ; 電源相序檢測異常
933   LDI     X10  ; 氣壓源壓力檢測
      AND     T7  ; 開機延遲5秒
      ANI     Y9  ; 進氣排水繼電器
      LD      M233  ; 氣壓源壓力檢測異常
      ANI     M9  ; 警報復歸PB
      ORB
      OUT     M233  ; 氣壓源壓力檢測異常
940   LD      X2  ; 溫控器 1加熱器異常
      AND     T7  ; 開機延遲5秒
      LD      M239  ; 溫控器 1加熱器異常
      ANI     M9  ; 警報復歸PB
      ORB
      MPS
      AND     T90  ; 溫控器 1加熱器異常TM
      OUT     M239  ; 溫控器 1加熱器異常
      MPP
      OUT     T90 K50  ; 溫控器 1加熱器異常TM
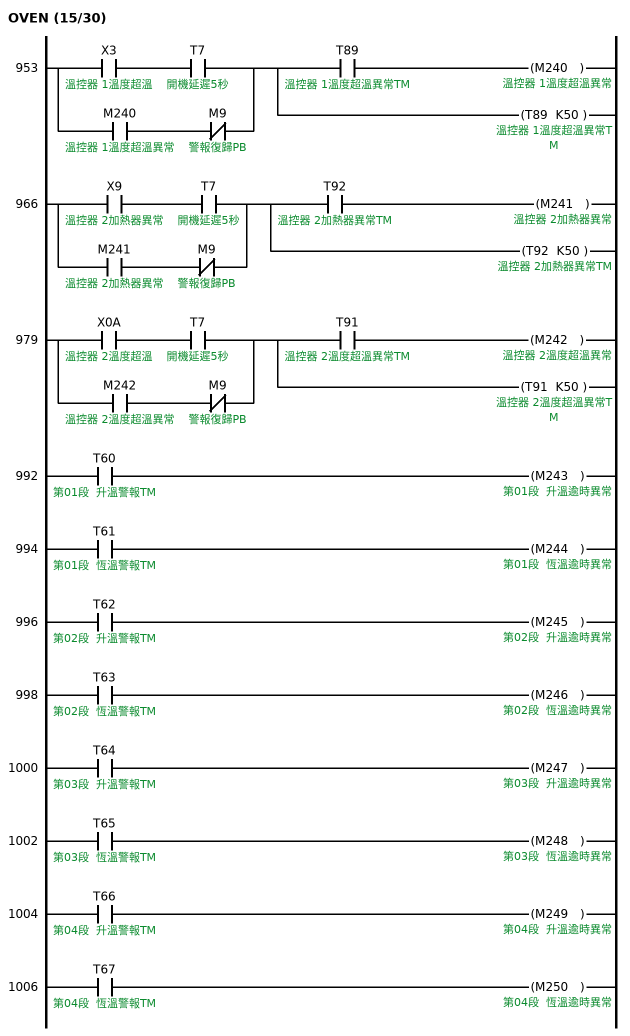
953   LD      X3  ; 溫控器 1溫度超溫
      AND     T7  ; 開機延遲5秒
      LD      M240  ; 溫控器 1溫度超溫異常
      ANI     M9  ; 警報復歸PB
      ORB
      MPS
      AND     T89  ; 溫控器 1溫度超溫異常TM
      OUT     M240  ; 溫控器 1溫度超溫異常
      MPP
      OUT     T89 K50  ; 溫控器 1溫度超溫異常TM
966   LD      X9  ; 溫控器 2加熱器異常
      AND     T7  ; 開機延遲5秒
      LD      M241  ; 溫控器 2加熱器異常
      ANI     M9  ; 警報復歸PB
      ORB
      MPS
      AND     T92  ; 溫控器 2加熱器異常TM
      OUT     M241  ; 溫控器 2加熱器異常
      MPP
      OUT     T92 K50  ; 溫控器 2加熱器異常TM
979   LD      X0A  ; 溫控器 2溫度超溫
      AND     T7  ; 開機延遲5秒
      LD      M242  ; 溫控器 2溫度超溫異常
      ANI     M9  ; 警報復歸PB
      ORB
      MPS
      AND     T91  ; 溫控器 2溫度超溫異常TM
      OUT     M242  ; 溫控器 2溫度超溫異常
      MPP
      OUT     T91 K50  ; 溫控器 2溫度超溫異常TM
992   LD      T60  ; 第01段  升溫警報TM
      OUT     M243  ; 第01段  升溫逾時異常
994   LD      T61  ; 第01段  恆溫警報TM
      OUT     M244  ; 第01段  恆溫逾時異常
996   LD      T62  ; 第02段  升溫警報TM
      OUT     M245  ; 第02段  升溫逾時異常
998   LD      T63  ; 第02段  恆溫警報TM
      OUT     M246  ; 第02段  恆溫逾時異常
1000  LD      T64  ; 第03段  升溫警報TM
      OUT     M247  ; 第03段  升溫逾時異常
1002  LD      T65  ; 第03段  恆溫警報TM
      OUT     M248  ; 第03段  恆溫逾時異常
1004  LD      T66  ; 第04段  升溫警報TM
      OUT     M249  ; 第04段  升溫逾時異常
1006  LD      T67  ; 第04段  恆溫警報TM
      OUT     M250  ; 第04段  恆溫逾時異常
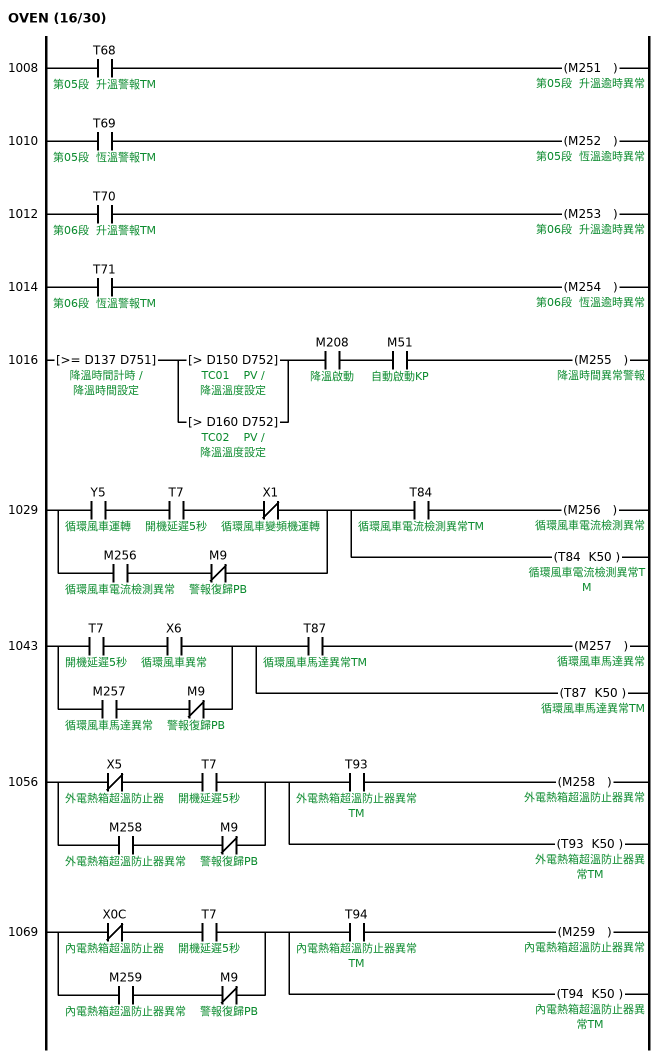
1008  LD      T68  ; 第05段  升溫警報TM
      OUT     M251  ; 第05段  升溫逾時異常
1010  LD      T69  ; 第05段  恆溫警報TM
      OUT     M252  ; 第05段  恆溫逾時異常
1012  LD      T70  ; 第06段  升溫警報TM
      OUT     M253  ; 第06段  升溫逾時異常
1014  LD      T71  ; 第06段  恆溫警報TM
      OUT     M254  ; 第06段  恆溫逾時異常
1016  LD>=    D137 D751  ; 降溫時間計時 / 降溫時間設定
      LD>     D150 D752  ; TC01    PV / 降溫溫度設定
      OR>     D160 D752  ; TC02    PV / 降溫溫度設定
      ANB
      AND     M208  ; 降溫啟動
      AND     M51  ; 自動啟動KP
      OUT     M255  ; 降溫時間異常警報
1029  LD      Y5  ; 循環風車運轉
      AND     T7  ; 開機延遲5秒
      ANI     X1  ; 循環風車變頻機運轉
      LD      M256  ; 循環風車電流檢測異常
      ANI     M9  ; 警報復歸PB
      ORB
      MPS
      AND     T84  ; 循環風車電流檢測異常TM
      OUT     M256  ; 循環風車電流檢測異常
      MPP
      OUT     T84 K50  ; 循環風車電流檢測異常TM
1043  LD      T7  ; 開機延遲5秒
      AND     X6  ; 循環風車異常
      LD      M257  ; 循環風車馬達異常
      ANI     M9  ; 警報復歸PB
      ORB
      MPS
      AND     T87  ; 循環風車馬達異常TM
      OUT     M257  ; 循環風車馬達異常
      MPP
      OUT     T87 K50  ; 循環風車馬達異常TM
1056  LDI     X5  ; 外電熱箱超溫防止器
      AND     T7  ; 開機延遲5秒
      LD      M258  ; 外電熱箱超溫防止器異常
      ANI     M9  ; 警報復歸PB
      ORB
      MPS
      AND     T93  ; 外電熱箱超溫防止器異常TM
      OUT     M258  ; 外電熱箱超溫防止器異常
      MPP
      OUT     T93 K50  ; 外電熱箱超溫防止器異常TM
1069  LDI     X0C  ; 內電熱箱超溫防止器
      AND     T7  ; 開機延遲5秒
      LD      M259  ; 內電熱箱超溫防止器異常
      ANI     M9  ; 警報復歸PB
      ORB
      MPS
      AND     T94  ; 內電熱箱超溫防止器異常TM
      OUT     M259  ; 內電熱箱超溫防止器異常
      MPP
      OUT     T94 K50  ; 內電熱箱超溫防止器異常TM
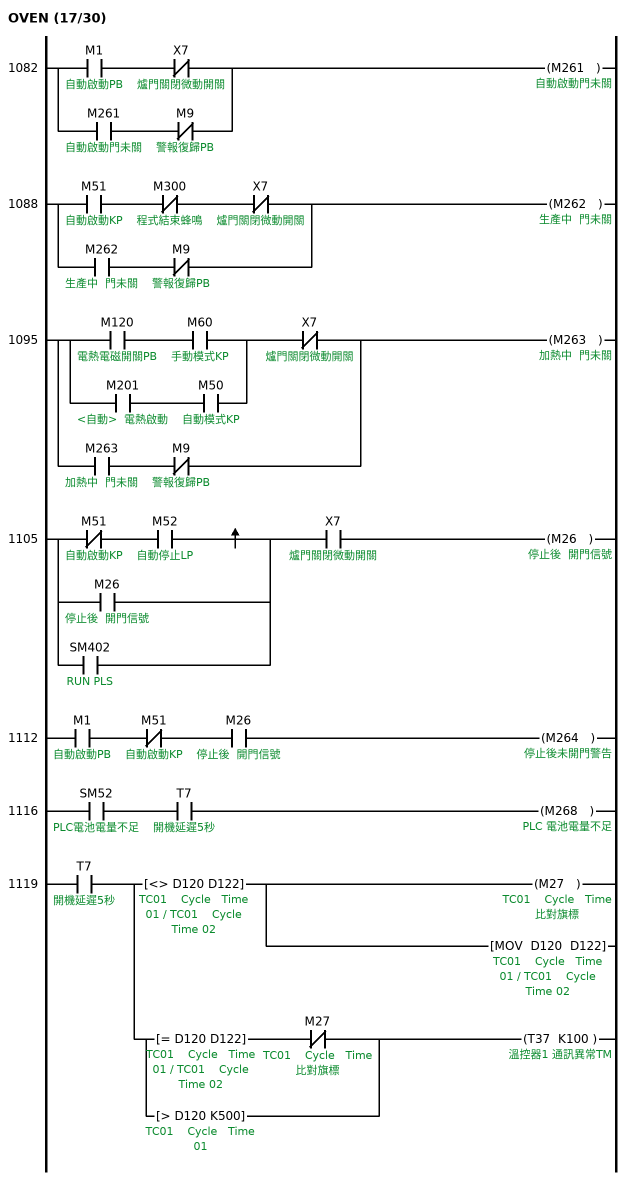
1082  LD      M1  ; 自動啟動PB
      ANI     X7  ; 爐門關閉微動開關
      LD      M261  ; 自動啟動門未關
      ANI     M9  ; 警報復歸PB
      ORB
      OUT     M261  ; 自動啟動門未關
1088  LD      M51  ; 自動啟動KP
      ANI     M300  ; 程式結束蜂鳴
      ANI     X7  ; 爐門關閉微動開關
      LD      M262  ; 生產中  門未關
      ANI     M9  ; 警報復歸PB
      ORB
      OUT     M262  ; 生產中  門未關
1095  LD      M120  ; 電熱電磁開關PB
      AND     M60  ; 手動模式KP
      LD      M201  ; <自動>  電熱啟動
      AND     M50  ; 自動模式KP
      ORB
      ANI     X7  ; 爐門關閉微動開關
      LD      M263  ; 加熱中  門未關
      ANI     M9  ; 警報復歸PB
      ORB
      OUT     M263  ; 加熱中  門未關
1105  LDI     M51  ; 自動啟動KP
      AND     M52  ; 自動停止LP
      MEP
      OR      M26  ; 停止後  開門信號
      OR      SM402  ; RUN PLS
      AND     X7  ; 爐門關閉微動開關
      OUT     M26  ; 停止後  開門信號
1112  LD      M1  ; 自動啟動PB
      ANI     M51  ; 自動啟動KP
      AND     M26  ; 停止後  開門信號
      OUT     M264  ; 停止後未開門警告
1116  LD      SM52  ; PLC電池電量不足
      AND     T7  ; 開機延遲5秒
      OUT     M268  ; PLC 電池電量不足
1119  LD      T7  ; 開機延遲5秒
      MPS
      AND<>   D120 D122  ; TC01    Cycle   Time 01 / TC01    Cycle   Time 02
      OUT     M27  ; TC01    Cycle   Time    比對旗標
      MOV     D120 D122
      MPP
      LD=     D120 D122  ; TC01    Cycle   Time 01 / TC01    Cycle   Time 02
      ANI     M27  ; TC01    Cycle   Time    比對旗標
      OR>     D120 K500  ; TC01    Cycle   Time 01
      ANB
      OUT     T37 K100  ; 溫控器1 通訊異常TM
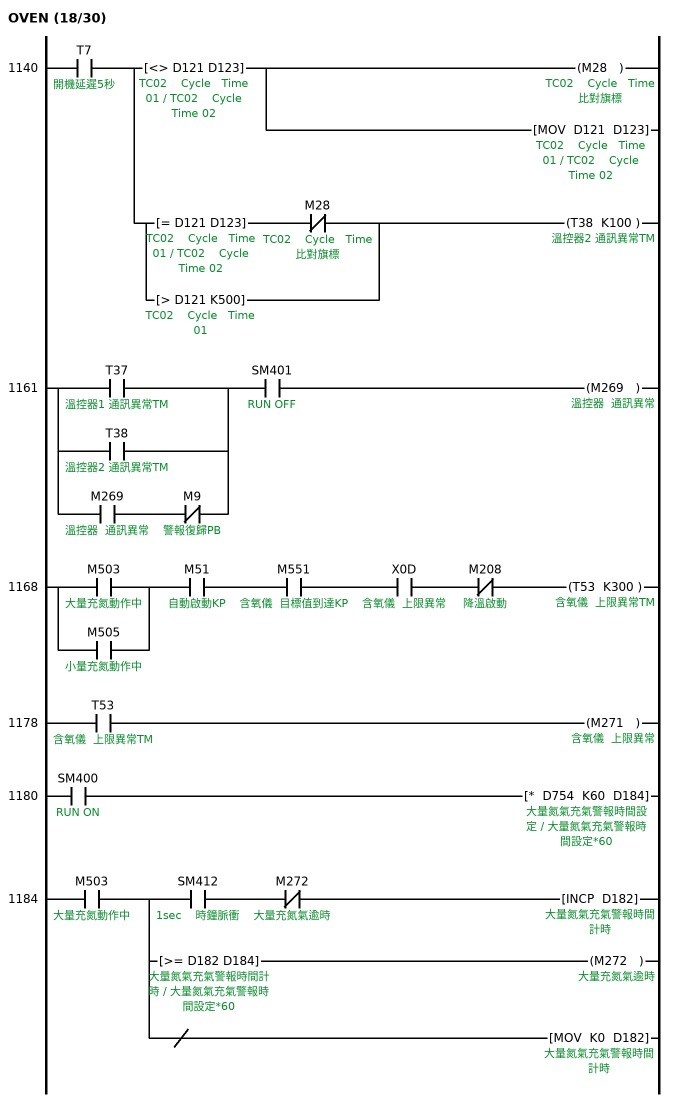
1140  LD      T7  ; 開機延遲5秒
      MPS
      AND<>   D121 D123  ; TC02    Cycle   Time 01 / TC02    Cycle   Time 02
      OUT     M28  ; TC02    Cycle   Time    比對旗標
      MOV     D121 D123
      MPP
      LD=     D121 D123  ; TC02    Cycle   Time 01 / TC02    Cycle   Time 02
      ANI     M28  ; TC02    Cycle   Time    比對旗標
      OR>     D121 K500  ; TC02    Cycle   Time 01
      ANB
      OUT     T38 K100  ; 溫控器2 通訊異常TM
1161  LD      T37  ; 溫控器1 通訊異常TM
      OR      T38  ; 溫控器2 通訊異常TM
      LD      M269  ; 溫控器  通訊異常
      ANI     M9  ; 警報復歸PB
      ORB
      AND     SM401  ; RUN OFF
      OUT     M269  ; 溫控器  通訊異常
1168  LD      M503  ; 大量充氮動作中
      OR      M505  ; 小量充氮動作中
      AND     M51  ; 自動啟動KP
      AND     M551  ; 含氧儀  目標值到達KP
      AND     X0D  ; 含氧儀  上限異常
      ANI     M208  ; 降溫啟動
      OUT     T53 K300  ; 含氧儀  上限異常TM
1178  LD      T53  ; 含氧儀  上限異常TM
      OUT     M271  ; 含氧儀  上限異常
1180  LD      SM400  ; RUN ON
      *       D754 K60 D184  ; 大量氮氣充氣警報時間設定 / 大量氮氣充氣警報時間設定*60
1184  LD      M503  ; 大量充氮動作中
      MPS
      AND     SM412  ; 1sec    時鐘脈衝
      ANI     M272  ; 大量充氮氣逾時
      INCP    D182  ; 大量氮氣充氣警報時間計時
      MRD
      AND>=   D182 D184  ; 大量氮氣充氣警報時間計時 / 大量氮氣充氣警報時間設定*60
      OUT     M272  ; 大量充氮氣逾時
      MPP
      INV
      MOV     K0 D182
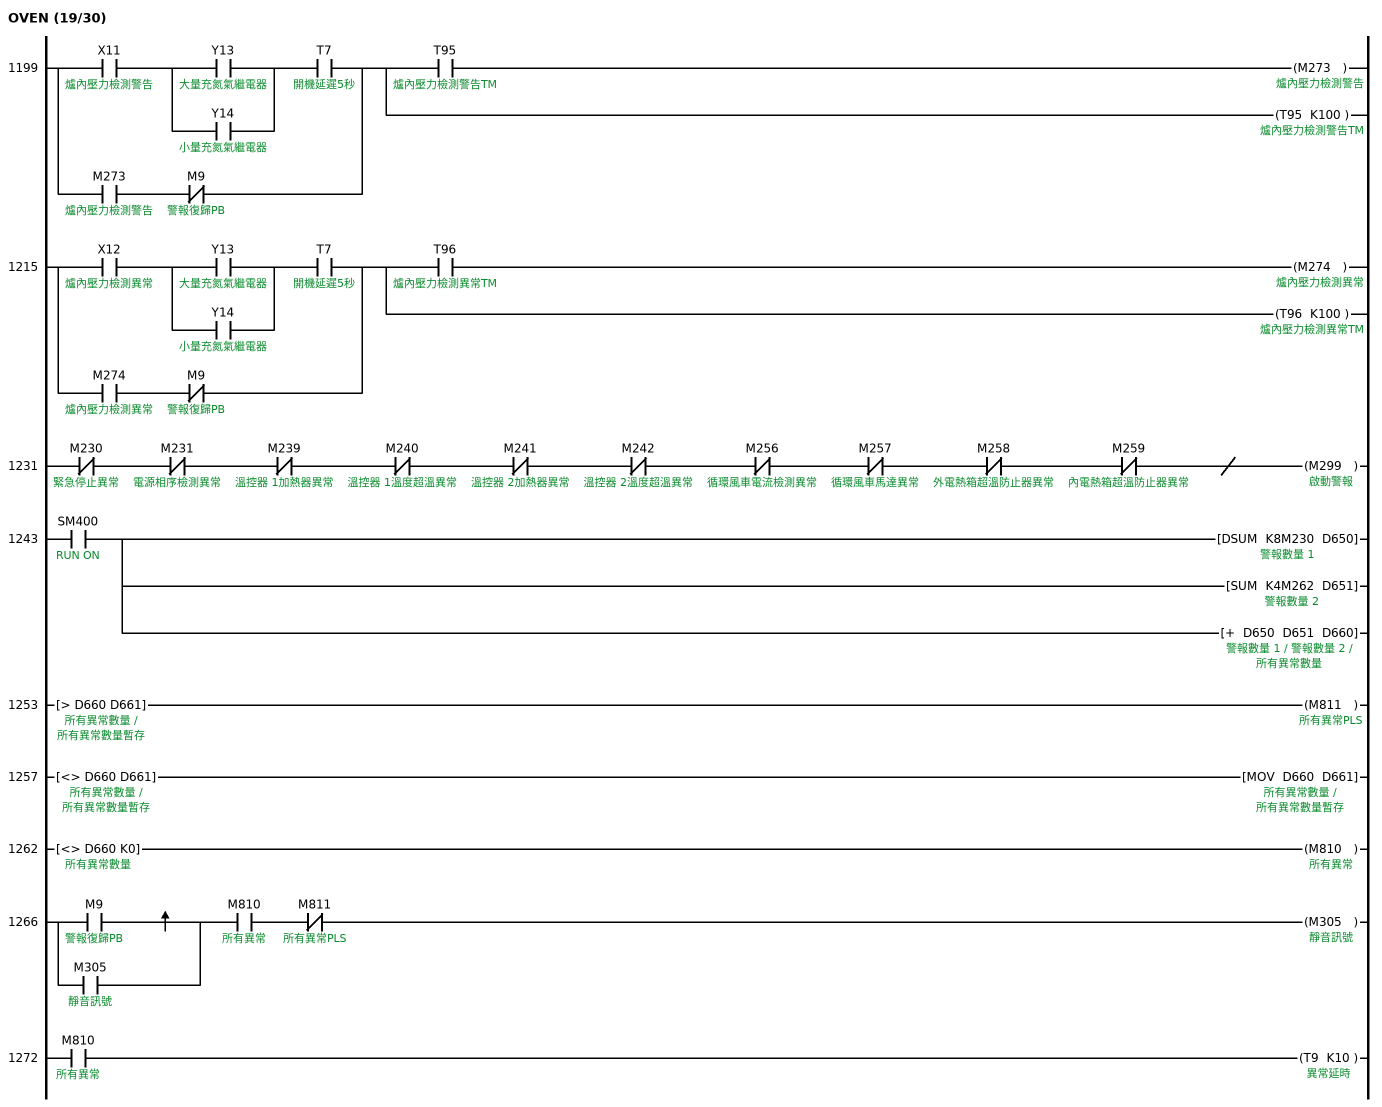
1199  LD      X11  ; 爐內壓力檢測警告
      LD      Y13  ; 大量充氮氣繼電器
      OR      Y14  ; 小量充氮氣繼電器
      ANB
      AND     T7  ; 開機延遲5秒
      LD      M273  ; 爐內壓力檢測警告
      ANI     M9  ; 警報復歸PB
      ORB
      MPS
      AND     T95  ; 爐內壓力檢測警告TM
      OUT     M273  ; 爐內壓力檢測警告
      MPP
      OUT     T95 K100  ; 爐內壓力檢測警告TM
1215  LD      X12  ; 爐內壓力檢測異常
      LD      Y13  ; 大量充氮氣繼電器
      OR      Y14  ; 小量充氮氣繼電器
      ANB
      AND     T7  ; 開機延遲5秒
      LD      M274  ; 爐內壓力檢測異常
      ANI     M9  ; 警報復歸PB
      ORB
      MPS
      AND     T96  ; 爐內壓力檢測異常TM
      OUT     M274  ; 爐內壓力檢測異常
      MPP
      OUT     T96 K100  ; 爐內壓力檢測異常TM
1231  LDI     M230  ; 緊急停止異常
      ANI     M231  ; 電源相序檢測異常
      ANI     M239  ; 溫控器 1加熱器異常
      ANI     M240  ; 溫控器 1溫度超溫異常
      ANI     M241  ; 溫控器 2加熱器異常
      ANI     M242  ; 溫控器 2溫度超溫異常
      ANI     M256  ; 循環風車電流檢測異常
      ANI     M257  ; 循環風車馬達異常
      ANI     M258  ; 外電熱箱超溫防止器異常
      ANI     M259  ; 內電熱箱超溫防止器異常
      INV
      OUT     M299  ; 啟動警報
1243  LD      SM400  ; RUN ON
      DSUM    K8M230 D650  ; 警報數量 1
      SUM     K4M262 D651  ; 警報數量 2
      +       D650 D651 D660  ; 所有異常數量
1253  LD>     D660 D661  ; 所有異常數量 / 所有異常數量暫存
      OUT     M811  ; 所有異常PLS
1257  LD<>    D660 D661  ; 所有異常數量 / 所有異常數量暫存
      MOV     D660 D661
1262  LD<>    D660 K0  ; 所有異常數量
      OUT     M810  ; 所有異常
1266  LD      M9  ; 警報復歸PB
      MEP
      OR      M305  ; 靜音訊號
      AND     M810  ; 所有異常
      ANI     M811  ; 所有異常PLS
      OUT     M305  ; 靜音訊號
1272  LD      M810  ; 所有異常
      OUT     T9 K10  ; 異常延時
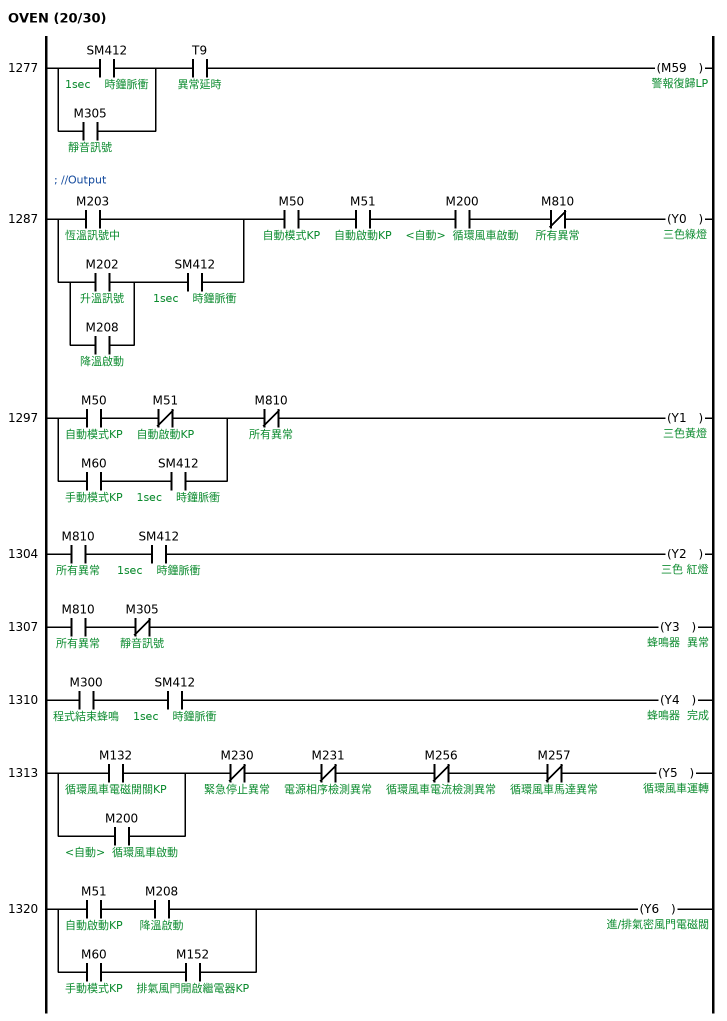
1277  LD      SM412  ; 1sec    時鐘脈衝
      OR      M305  ; 靜音訊號
      AND     T9  ; 異常延時
      OUT     M59  ; 警報復歸LP
; //Output
1287  LD      M203  ; 恆溫訊號中
      LD      M202  ; 升溫訊號
      OR      M208  ; 降溫啟動
      AND     SM412  ; 1sec    時鐘脈衝
      ORB
      AND     M50  ; 自動模式KP
      AND     M51  ; 自動啟動KP
      AND     M200  ; <自動>  循環風車啟動
      ANI     M810  ; 所有異常
      OUT     Y0  ; 三色綠燈
1297  LD      M50  ; 自動模式KP
      ANI     M51  ; 自動啟動KP
      LD      M60  ; 手動模式KP
      AND     SM412  ; 1sec    時鐘脈衝
      ORB
      ANI     M810  ; 所有異常
      OUT     Y1  ; 三色黃燈
1304  LD      M810  ; 所有異常
      AND     SM412  ; 1sec    時鐘脈衝
      OUT     Y2  ; 三色 紅燈
1307  LD      M810  ; 所有異常
      ANI     M305  ; 靜音訊號
      OUT     Y3  ; 蜂鳴器  異常
1310  LD      M300  ; 程式結束蜂鳴
      AND     SM412  ; 1sec    時鐘脈衝
      OUT     Y4  ; 蜂鳴器  完成
1313  LD      M132  ; 循環風車電磁開關KP
      OR      M200  ; <自動>  循環風車啟動
      ANI     M230  ; 緊急停止異常
      ANI     M231  ; 電源相序檢測異常
      ANI     M256  ; 循環風車電流檢測異常
      ANI     M257  ; 循環風車馬達異常
      OUT     Y5  ; 循環風車運轉
1320  LD      M51  ; 自動啟動KP
      AND     M208  ; 降溫啟動
      LD      M60  ; 手動模式KP
      AND     M152  ; 排氣風門開啟繼電器KP
      ORB
      OUT     Y6  ; 進/排氣密風門電磁閥
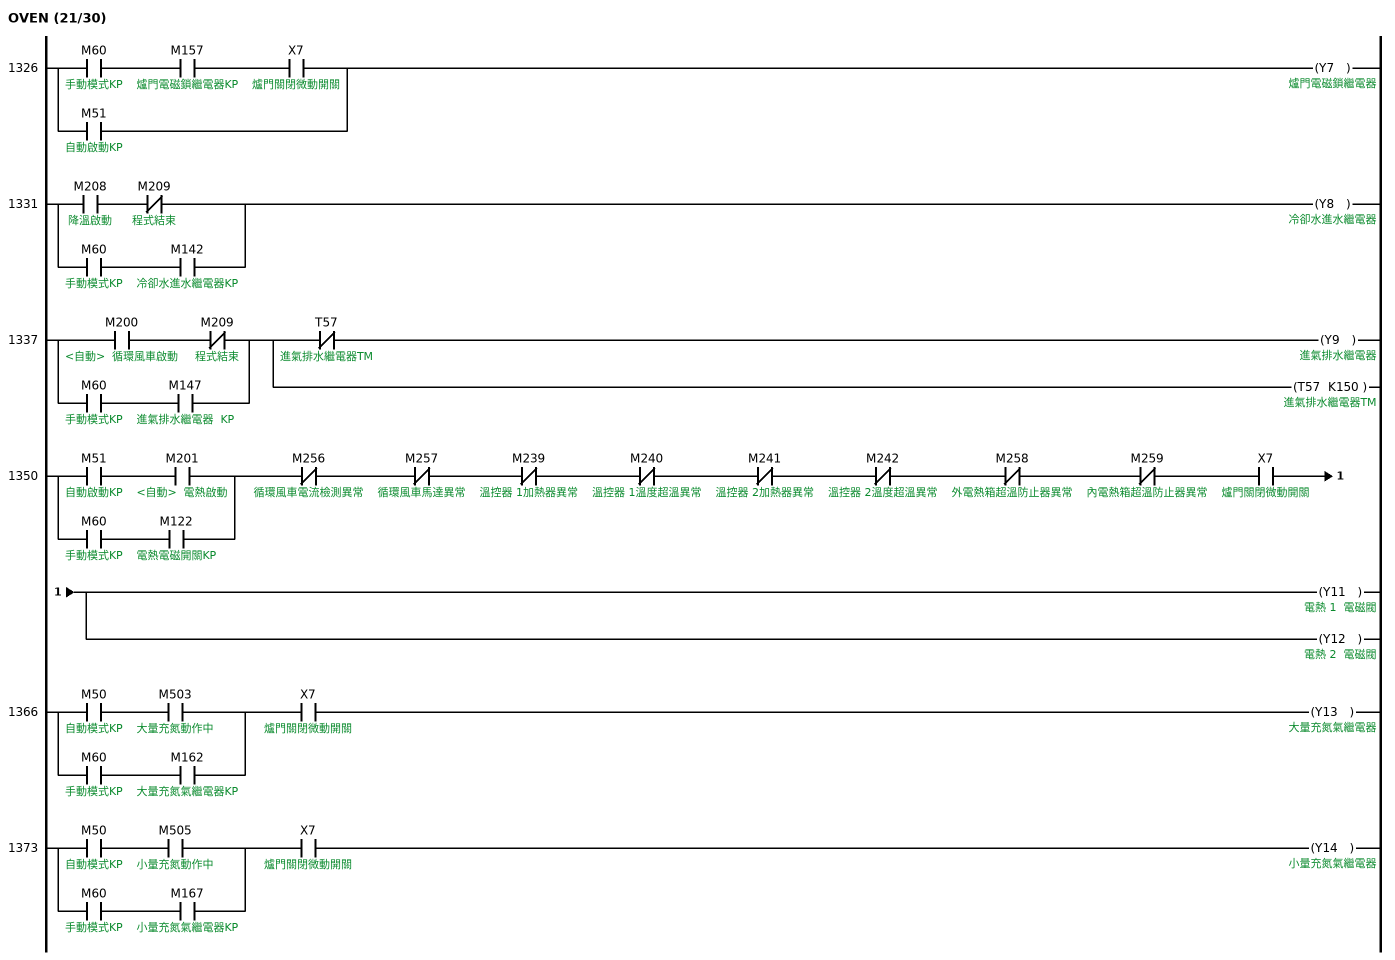
1326  LD      M60  ; 手動模式KP
      AND     M157  ; 爐門電磁鎖繼電器KP
      AND     X7  ; 爐門關閉微動開關
      OR      M51  ; 自動啟動KP
      OUT     Y7  ; 爐門電磁鎖繼電器
1331  LD      M208  ; 降溫啟動
      ANI     M209  ; 程式結束
      LD      M60  ; 手動模式KP
      AND     M142  ; 冷卻水進水繼電器KP
      ORB
      OUT     Y8  ; 冷卻水進水繼電器
1337  LD      M200  ; <自動>  循環風車啟動
      ANI     M209  ; 程式結束
      LD      M60  ; 手動模式KP
      AND     M147  ; 進氣排水繼電器  KP
      ORB
      MPS
      ANI     T57  ; 進氣排水繼電器TM
      OUT     Y9  ; 進氣排水繼電器
      MPP
      OUT     T57 K150  ; 進氣排水繼電器TM
1350  LD      M51  ; 自動啟動KP
      AND     M201  ; <自動>  電熱啟動
      LD      M60  ; 手動模式KP
      AND     M122  ; 電熱電磁開關KP
      ORB
      ANI     M256  ; 循環風車電流檢測異常
      ANI     M257  ; 循環風車馬達異常
      ANI     M239  ; 溫控器 1加熱器異常
      ANI     M240  ; 溫控器 1溫度超溫異常
      ANI     M241  ; 溫控器 2加熱器異常
      ANI     M242  ; 溫控器 2溫度超溫異常
      ANI     M258  ; 外電熱箱超溫防止器異常
      ANI     M259  ; 內電熱箱超溫防止器異常
      AND     X7  ; 爐門關閉微動開關
      OUT     Y11  ; 電熱 1  電磁閥
      OUT     Y12  ; 電熱 2  電磁閥
1366  LD      M50  ; 自動模式KP
      AND     M503  ; 大量充氮動作中
      LD      M60  ; 手動模式KP
      AND     M162  ; 大量充氮氣繼電器KP
      ORB
      AND     X7  ; 爐門關閉微動開關
      OUT     Y13  ; 大量充氮氣繼電器
1373  LD      M50  ; 自動模式KP
      AND     M505  ; 小量充氮動作中
      LD      M60  ; 手動模式KP
      AND     M167  ; 小量充氮氣繼電器KP
      ORB
      AND     X7  ; 爐門關閉微動開關
      OUT     Y14  ; 小量充氮氣繼電器
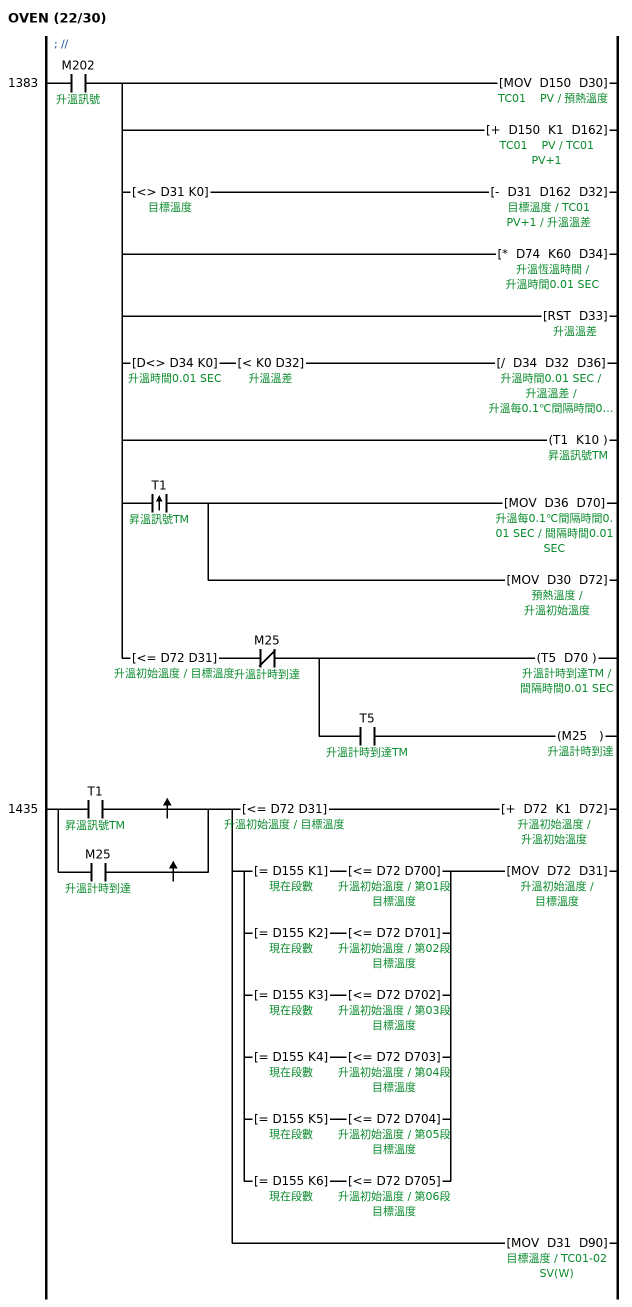
; //
1383  LD      M202  ; 升溫訊號
      MOV     D150 D30  ; 預熱溫度
      +       D150 K1 D162  ; TC01    PV+1
      MPS
      AND<>   D31 K0  ; 目標溫度
      -       D31 D162 D32  ; 升溫溫差
      MPP
      *       D74 K60 D34  ; 升溫時間0.01 SEC
      RST     D33  ; 升溫溫差
      MPS
      ANDD<>  D34 K0  ; 升溫時間0.01 SEC
      AND<    K0 D32  ; 升溫溫差
      /       D34 D32 D36  ; 升溫每0.1℃間隔時間0.01 SEC
      MPP
      OUT     T1 K10  ; 昇溫訊號TM
      MPS
      ANDP    T1  ; 昇溫訊號TM
      MOV     D36 D70  ; 間隔時間0.01 SEC
      MOV     D30 D72
      MPP
      AND<=   D72 D31  ; 升溫初始溫度 / 目標溫度
      ANI     M25  ; 升溫計時到達
      OUT     T5 D70  ; 升溫計時到達TM / 間隔時間0.01 SEC
      AND     T5  ; 升溫計時到達TM
      OUT     M25  ; 升溫計時到達
1435  LD      T1  ; 昇溫訊號TM
      MEP
      LD      M25  ; 升溫計時到達
      MEP
      ORB
      MPS
      AND<=   D72 D31  ; 升溫初始溫度 / 目標溫度
      +       D72 K1 D72
      MRD
      LD=     D155 K1  ; 現在段數
      AND<=   D72 D700  ; 升溫初始溫度 / 第01段  目標溫度
      LD=     D155 K2  ; 現在段數
      AND<=   D72 D701  ; 升溫初始溫度 / 第02段  目標溫度
      ORB
      LD=     D155 K3  ; 現在段數
      AND<=   D72 D702  ; 升溫初始溫度 / 第03段  目標溫度
      ORB
      LD=     D155 K4  ; 現在段數
      AND<=   D72 D703  ; 升溫初始溫度 / 第04段  目標溫度
      ORB
      LD=     D155 K5  ; 現在段數
      AND<=   D72 D704  ; 升溫初始溫度 / 第05段  目標溫度
      ORB
      LD=     D155 K6  ; 現在段數
      AND<=   D72 D705  ; 升溫初始溫度 / 第06段  目標溫度
      ORB
      ANB
      MOV     D72 D31
      MPP
      MOV     D31 D90  ; TC01-02 SV(W)
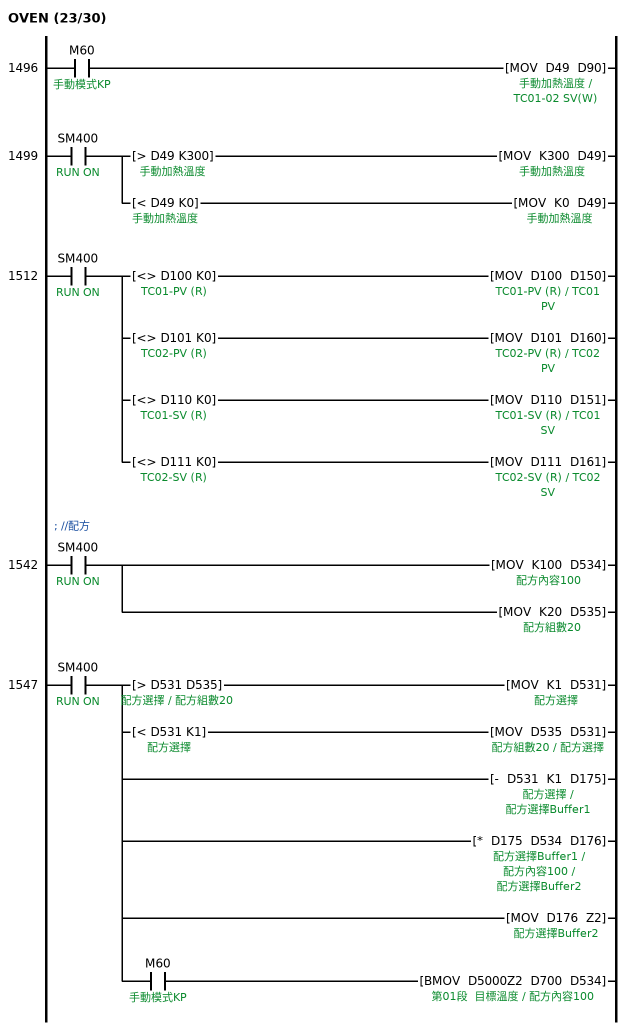
1496  LD      M60  ; 手動模式KP
      MOV     D49 D90  ; 手動加熱溫度
1499  LD      SM400  ; RUN ON
      MPS
      AND>    D49 K300  ; 手動加熱溫度
      MOV     K300 D49
      MPP
      AND<    D49 K0  ; 手動加熱溫度
      MOV     K0 D49
1512  LD      SM400  ; RUN ON
      MPS
      AND<>   D100 K0  ; TC01-PV (R)
      MOV     D100 D150
      MRD
      AND<>   D101 K0  ; TC02-PV (R)
      MOV     D101 D160
      MRD
      AND<>   D110 K0  ; TC01-SV (R)
      MOV     D110 D151  ; TC01    SV
      MPP
      AND<>   D111 K0  ; TC02-SV (R)
      MOV     D111 D161  ; TC02    SV
; //配方
1542  LD      SM400  ; RUN ON
      MOV     K100 D534  ; 配方內容100
      MOV     K20 D535  ; 配方組數20
1547  LD      SM400  ; RUN ON
      MPS
      AND>    D531 D535  ; 配方選擇 / 配方組數20
      MOV     K1 D531
      MRD
      AND<    D531 K1  ; 配方選擇
      MOV     D535 D531
      MPP
      -       D531 K1 D175  ; 配方選擇Buffer1
      *       D175 D534 D176  ; 配方選擇Buffer2
      MOV     D176 Z2
      AND     M60  ; 手動模式KP
      BMOV    D5000Z2 D700 D534
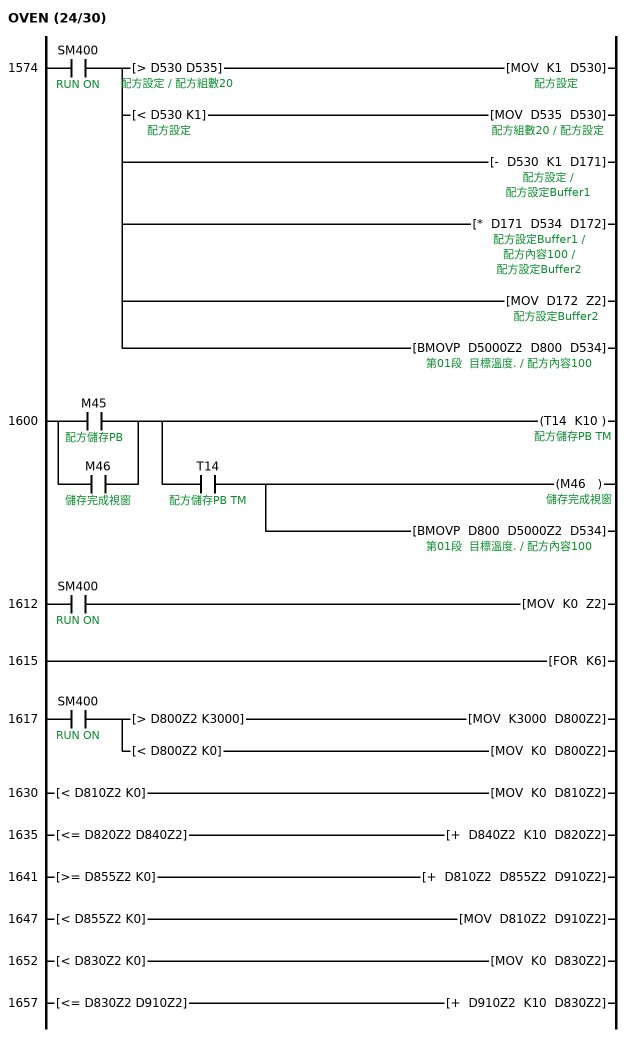
1574  LD      SM400  ; RUN ON
      MPS
      AND>    D530 D535  ; 配方設定 / 配方組數20
      MOV     K1 D530
      MRD
      AND<    D530 K1  ; 配方設定
      MOV     D535 D530
      MPP
      -       D530 K1 D171  ; 配方設定Buffer1
      *       D171 D534 D172  ; 配方設定Buffer2
      MOV     D172 Z2
      BMOVP   D5000Z2 D800 D534  ; 第01段  目標溫度.
1600  LD      M45  ; 配方儲存PB
      OR      M46  ; 儲存完成視窗
      OUT     T14 K10  ; 配方儲存PB TM
      AND     T14  ; 配方儲存PB TM
      OUT     M46  ; 儲存完成視窗
      BMOVP   D800 D5000Z2 D534
1612  LD      SM400  ; RUN ON
      MOV     K0 Z2
1615  FOR     K6
1617  LD      SM400  ; RUN ON
      MPS
      AND>    D800Z2 K3000
      MOV     K3000 D800Z2
      MPP
      AND<    D800Z2 K0
      MOV     K0 D800Z2
1630  LD<     D810Z2 K0
      MOV     K0 D810Z2
1635  LD<=    D820Z2 D840Z2
      +       D840Z2 K10 D820Z2
1641  LD>=    D855Z2 K0
      +       D810Z2 D855Z2 D910Z2
1647  LD<     D855Z2 K0
      MOV     D810Z2 D910Z2
1652  LD<     D830Z2 K0
      MOV     K0 D830Z2
1657  LD<=    D830Z2 D910Z2
      +       D910Z2 K10 D830Z2
